LIN {X 0,Y 389.077,Z 656.988,A -85,B 0,C 180,E1 10601.483,E2 10601.483} C_VEL
LIN {X 0,Y 373.239,Z 818.988,A -85,B 0,C 180,E1 10598.992,E2 10598.992} C_VEL
LIN {X 0,Y 369.039,Z 845.316,A -85,B 0,C 180,E1 10598.451,E2 10598.451} C_VEL
LIN {X 0,Y 364.552,Z 865.956,A -85,B 0,C 180,E1 10597.891,E2 10597.891} C_VEL
LIN {X 0,Y 357.971,Z 890.119,A -85,B 0,C 180,E1 10597.055,E2 10597.055} C_VEL
LIN {X 0,Y 350.974,Z 911.054,A -85,B 0,C 180,E1 10596.135,E2 10596.135} C_VEL
LIN {X 0,Y 342.625,Z 932.727,A -85,B 0,C 180,E1 10594.966,E2 10594.966} C_VEL
LIN {X 0,Y 332.858,Z 954.168,A -85,B 0,C 180,E1 10593.532,E2 10593.532} C_VEL
LIN {X 0,Y 322.694,Z 974.134,A -85,B 0,C 180,E1 10591.902,E2 10591.902} C_VEL
LIN {X 0,Y 311.477,Z 993.542,A -85,B 0,C 180,E1 10589.948,E2 10589.948} C_VEL
LIN {X 0,Y 300.928,Z 1010.196,A -85,B 0,C 180,E1 10587.918,E2 10587.918} C_VEL
LIN {X 0,Y 287.781,Z 1029.047,A -85,B 0,C 180,E1 10585.083,E2 10585.083} C_VEL
LIN {X 0,Y 276.633,Z 1043.791,A -85,B 0,C 180,E1 10582.333,E2 10582.333} C_VEL
LIN {X 0,Y 263.742,Z 1059.682,A -85,B 0,C 180,E1 10578.647,E2 10578.647} C_VEL
LIN {X 0,Y 253.035,Z 1072.129,A -85,B 0,C 180,E1 10575.019,E2 10575.019} C_VEL
LIN {X 0,Y 241.418,Z 1085.134,A -85,B 0,C 180,E1 10570.249,E2 10570.249} C_VEL
LIN {X 0,Y 232.232,Z 1095.159,A -85,B 0,C 180,E1 10565.539,E2 10565.539} C_VEL
LIN {X 0,Y 223.527,Z 1104.789,A -85,B 0,C 180,E1 10559.771,E2 10559.771} C_VEL
LIN {X 0,Y 217.336,Z 1111.9,A -85,B 0,C 180,E1 10554.171,E2 10554.171} C_VEL
LIN {X 0,Y 212.563,Z 1118.125,A -85,B 0,C 180,E1 10547.804,E2 10547.804} C_VEL
LIN {X 0,Y 209.773,Z 1122.382,A -85,B 0,C 180,E1 10541.548,E2 10541.548} C_VEL
LIN {X 0,Y 208.571,Z 1124.988,A -85,B 0,C 180,E1 10536.054,E2 10536.054} C_VEL
LIN {X 0,Y 208.165,Z 1126.701,A -85,B 0,C 180,E1 10530,E2 10530} C_VEL
LIN {X 0,Y 208.154,Z 1127.046,A -85,B 0,C 180,E1 10524.21,E2 10524.21} C_VEL
LIN {X 0,Y 208.486,Z 1126.397,A -85,B 0,C 180,E1 10518.94,E2 10518.94} C_VEL
LIN {X 0,Y 209.585,Z 1124.699,A -85,B 0,C 180,E1 10513.366,E2 10513.366} C_VEL
LIN {X 0,Y 212.305,Z 1121.48,A -85,B 0,C 180,E1 10506.989,E2 10506.989} C_VEL
LIN {X 0,Y 217.097,Z 1116.332,A -85,B 0,C 180,E1 10500.474,E2 10500.474} C_VEL
LIN {X 0,Y 223.889,Z 1109.804,A -85,B 0,C 180,E1 10494.372,E2 10494.372} C_VEL
LIN {X 0,Y 232.384,Z 1101.701,A -85,B 0,C 180,E1 10488.828,E2 10488.828} C_VEL
LIN {X 0,Y 241.918,Z 1092.689,A -85,B 0,C 180,E1 10484.013,E2 10484.013} C_VEL
LIN {X 0,Y 254.032,Z 1080.851,A -85,B 0,C 180,E1 10479.158,E2 10479.158} C_VEL
LIN {X 0,Y 265.219,Z 1069.449,A -85,B 0,C 180,E1 10475.478,E2 10475.478} C_VEL
LIN {X 0,Y 278.682,Z 1054.854,A -85,B 0,C 180,E1 10471.751,E2 10471.751} C_VEL
LIN {X 0,Y 290.339,Z 1041.264,A -85,B 0,C 180,E1 10468.985,E2 10468.985} C_VEL
LIN {X 0,Y 303.745,Z 1024.447,A -85,B 0,C 180,E1 10466.207,E2 10466.207} C_VEL
LIN {X 0,Y 315.589,Z 1008.029,A -85,B 0,C 180,E1 10464.034,E2 10464.034} C_VEL
LIN {X 0,Y 327.873,Z 989.488,A -85,B 0,C 180,E1 10462.014,E2 10462.014} C_VEL
LIN {X 0,Y 339.512,Z 969.544,A -85,B 0,C 180,E1 10460.266,E2 10460.266} C_VEL
LIN {X 0,Y 349.337,Z 950.846,A -85,B 0,C 180,E1 10458.919,E2 10458.919} C_VEL
LIN {X 0,Y 359.347,Z 928.996,A -85,B 0,C 180,E1 10457.633,E2 10457.633} C_VEL
LIN {X 0,Y 366.943,Z 909.841,A -85,B 0,C 180,E1 10456.702,E2 10456.702} C_VEL
LIN {X 0,Y 374.785,Z 886.816,A -85,B 0,C 180,E1 10455.791,E2 10455.791} C_VEL
LIN {X 0,Y 381.061,Z 863.843,A -85,B 0,C 180,E1 10455.085,E2 10455.085} C_VEL
LIN {X 0,Y 386.288,Z 839.912,A -85,B 0,C 180,E1 10454.513,E2 10454.513} C_VEL
LIN {X 0,Y 389.922,Z 815.583,A -85,B 0,C 180,E1 10454.078,E2 10454.078} C_VEL
LIN {X 0,Y 404.87,Z 668.819,A -85,B 0,C 180,E1 10451.908,E2 10451.908} C_VEL
LIN {X 0,Y 401.866,Z 662.718,A -85,B 0,C 180,E1 10449.38,E2 10449.38} C_VEL
LIN {X 0,Y 400.205,Z 659.502,A -85,B 0,C 180,E1 10447.682,E2 10447.682} C_VEL
LIN {X 0,Y 398.698,Z 656.415,A -85,B 0,C 180,E1 10445.757,E2 10445.757} C_VEL
LIN {X 0,Y 396.955,Z 652.484,A -85,B 0,C 180,E1 10442.31,E2 10442.31} C_VEL
LIN {X 0,Y 396.309,Z 651.938,A -85,B 0,C 180,E1 10437.686,E2 10437.686} C_VEL
LIN {X 0,Y 397.092,Z 652.674,A -85,B 0,C 180,E1 10434.799,E2 10434.799} C_VEL
LIN {X 0,Y 397.231,Z 653.236,A -85,B 0,C 180,E1 10434.385,E2 10434.385} C_VEL
LIN {X 0,Y 397.569,Z 655.643,A -85,B 0,C 180,E1 10433.318,E2 10433.318} C_VEL
LIN {X 0,Y 398.682,Z 666,A -85,B 0,C 180,E1 10430.456,E2 10430.456} C_VEL
LIN {X 0,Y 399.282,Z 667.678,A -85,B 0,C 180,E1 10429.696,E2 10429.696} C_VEL
LIN {X 0,Y 401.751,Z 672.925,A -85,B 0,C 180,E1 10427.239,E2 10427.239} C_VEL
LIN {X 0,Y 402.563,Z 675.356,A -85,B 0,C 180,E1 10426.485,E2 10426.485} C_VEL
LIN {X 0,Y 386.785,Z 826.745,A -85,B 0,C 180,E1 10424.281,E2 10424.281} C_VEL
LIN {X 0,Y 382.278,Z 853.306,A -85,B 0,C 180,E1 10423.81,E2 10423.81} C_VEL
LIN {X 0,Y 377.108,Z 875.277,A -85,B 0,C 180,E1 10423.339,E2 10423.339} C_VEL
LIN {X 0,Y 369.772,Z 899.868,A -85,B 0,C 180,E1 10422.658,E2 10422.658} C_VEL
LIN {X 0,Y 362.204,Z 920.785,A -85,B 0,C 180,E1 10421.909,E2 10421.909} C_VEL
LIN {X 0,Y 352.874,Z 943.017,A -85,B 0,C 180,E1 10420.908,E2 10420.908} C_VEL
LIN {X 0,Y 343.111,Z 962.976,A -85,B 0,C 180,E1 10419.78,E2 10419.78} C_VEL
LIN {X 0,Y 332.272,Z 982.798,A -85,B 0,C 180,E1 10418.414,E2 10418.414} C_VEL
LIN {X 0,Y 320.029,Z 1002.552,A -85,B 0,C 180,E1 10416.718,E2 10416.718} C_VEL
LIN {X 0,Y 308.525,Z 1019.414,A -85,B 0,C 180,E1 10414.935,E2 10414.935} C_VEL
LIN {X 0,Y 294.339,Z 1038.307,A -85,B 0,C 180,E1 10412.454,E2 10412.454} C_VEL
LIN {X 0,Y 281.858,Z 1053.497,A -85,B 0,C 180,E1 10409.95,E2 10409.95} C_VEL
LIN {X 0,Y 267.962,Z 1069.274,A -85,B 0,C 180,E1 10406.705,E2 10406.705} C_VEL
LIN {X 0,Y 255.148,Z 1082.75,A -85,B 0,C 180,E1 10403.16,E2 10403.16} C_VEL
LIN {X 0,Y 242.608,Z 1095.445,A -85,B 0,C 180,E1 10398.958,E2 10398.958} C_VEL
LIN {X 0,Y 231.059,Z 1106.532,A -85,B 0,C 180,E1 10394.164,E2 10394.164} C_VEL
LIN {X 0,Y 220.814,Z 1116.462,A -85,B 0,C 180,E1 10388.674,E2 10388.674} C_VEL
LIN {X 0,Y 212.27,Z 1124.783,A -85,B 0,C 180,E1 10382.479,E2 10382.479} C_VEL
LIN {X 0,Y 206.062,Z 1131.495,A -85,B 0,C 180,E1 10375.895,E2 10375.895} C_VEL
LIN {X 0,Y 202.161,Z 1136.355,A -85,B 0,C 180,E1 10369.053,E2 10369.053} C_VEL
LIN {X 0,Y 200.522,Z 1139.217,A -85,B 0,C 180,E1 10363.26,E2 10363.26} C_VEL
LIN {X 0,Y 200.045,Z 1141.13,A -85,B 0,C 180,E1 10356.89,E2 10356.89} C_VEL
LIN {X 0,Y 200.113,Z 1141.605,A -85,B 0,C 180,E1 10351.432,E2 10351.432} C_VEL
LIN {X 0,Y 200.082,Z 1141.072,A -85,B 0,C 180,E1 10346.275,E2 10346.275} C_VEL
LIN {X 0,Y 200.105,Z 1139.478,A -85,B 0,C 180,E1 10340.799,E2 10340.799} C_VEL
LIN {X 0,Y 200.858,Z 1136.684,A -85,B 0,C 180,E1 10334.997,E2 10334.997} C_VEL
LIN {X 0,Y 203.257,Z 1132.107,A -85,B 0,C 180,E1 10328.349,E2 10328.349} C_VEL
LIN {X 0,Y 207.889,Z 1125.467,A -85,B 0,C 180,E1 10321.565,E2 10321.565} C_VEL
LIN {X 0,Y 214.178,Z 1117.89,A -85,B 0,C 180,E1 10315.605,E2 10315.605} C_VEL
LIN {X 0,Y 222.875,Z 1108.056,A -85,B 0,C 180,E1 10309.701,E2 10309.701} C_VEL
LIN {X 0,Y 231.964,Z 1098.075,A -85,B 0,C 180,E1 10304.986,E2 10304.986} C_VEL
LIN {X 0,Y 244.099,Z 1084.603,A -85,B 0,C 180,E1 10300.004,E2 10300.004} C_VEL
LIN {X 0,Y 254.771,Z 1072.356,A -85,B 0,C 180,E1 10296.432,E2 10296.432} C_VEL
LIN {X 0,Y 267.773,Z 1056.749,A -85,B 0,C 180,E1 10292.782,E2 10292.782} C_VEL
LIN {X 0,Y 279.395,Z 1041.739,A -85,B 0,C 180,E1 10289.995,E2 10289.995} C_VEL
LIN {X 0,Y 292.125,Z 1024.23,A -85,B 0,C 180,E1 10287.349,E2 10287.349} C_VEL
LIN {X 0,Y 304.257,Z 1005.693,A -85,B 0,C 180,E1 10285.124,E2 10285.124} C_VEL
LIN {X 0,Y 315.234,Z 987.407,A -85,B 0,C 180,E1 10283.325,E2 10283.325} C_VEL
LIN {X 0,Y 326.531,Z 966.324,A -85,B 0,C 180,E1 10281.663,E2 10281.663} C_VEL
LIN {X 0,Y 336.004,Z 946.38,A -85,B 0,C 180,E1 10280.382,E2 10280.382} C_VEL
LIN {X 0,Y 345.665,Z 922.993,A -85,B 0,C 180,E1 10279.186,E2 10279.186} C_VEL
LIN {X 0,Y 352.927,Z 902.419,A -85,B 0,C 180,E1 10278.358,E2 10278.358} C_VEL
LIN {X 0,Y 360.033,Z 878.466,A -85,B 0,C 180,E1 10277.598,E2 10277.598} C_VEL
LIN {X 0,Y 365.3,Z 855.714,A -85,B 0,C 180,E1 10277.045,E2 10277.045} C_VEL
LIN {X 0,Y 369.595,Z 830.946,A -85,B 0,C 180,E1 10276.554,E2 10276.554} C_VEL
LIN {X 0,Y 375.172,Z 776.826,A -85,B 0,C 180,E1 10275.706,E2 10275.706} C_VEL
LIN {X 0,Y 386.379,Z 662.671,A -85,B 0,C 180,E1 10273.975,E2 10273.975} C_VEL
LIN {X 0,Y 384.218,Z 657.456,A -85,B 0,C 180,E1 10272.398,E2 10272.398} C_VEL
LIN {X 0,Y 380.921,Z 650.9,A -85,B 0,C 180,E1 10269.671,E2 10269.671} C_VEL
LIN {X 0,Y 378.814,Z 646.848,A -85,B 0,C 180,E1 10267.508,E2 10267.508} C_VEL
LIN {X 0,Y 377.258,Z 643.74,A -85,B 0,C 180,E1 10265.475,E2 10265.475} C_VEL
LIN {X 0,Y 375.486,Z 639.736,A -85,B 0,C 180,E1 10261.831,E2 10261.831} C_VEL
LIN {X 0,Y 374.913,Z 639.355,A -85,B 0,C 180,E1 10256.789,E2 10256.789} C_VEL
LIN {X 0,Y 375.595,Z 640.112,A -85,B 0,C 180,E1 10254.271,E2 10254.271} C_VEL
LIN {X 0,Y 377.781,Z 644.756,A -85,B 0,C 180,E1 10250.247,E2 10250.247} C_VEL
LIN {X 0,Y 380.132,Z 649.399,A -85,B 0,C 180,E1 10247.544,E2 10247.544} C_VEL
LIN {X 0,Y 382.994,Z 654.95,A -85,B 0,C 180,E1 10245.01,E2 10245.01} C_VEL
LIN {X 0,Y 386.347,Z 662.03,A -85,B 0,C 180,E1 10242.546,E2 10242.546} C_VEL
LIN {X 0,Y 370.657,Z 819.269,A -85,B 0,C 180,E1 10240.158,E2 10240.158} C_VEL
LIN {X 0,Y 366.382,Z 845.61,A -85,B 0,C 180,E1 10239.627,E2 10239.627} C_VEL
LIN {X 0,Y 361.82,Z 866.249,A -85,B 0,C 180,E1 10239.078,E2 10239.078} C_VEL
LIN {X 0,Y 355.206,Z 890.16,A -85,B 0,C 180,E1 10238.27,E2 10238.27} C_VEL
LIN {X 0,Y 347.96,Z 911.47,A -85,B 0,C 180,E1 10237.352,E2 10237.352} C_VEL
LIN {X 0,Y 339.387,Z 933.291,A -85,B 0,C 180,E1 10236.195,E2 10236.195} C_VEL
LIN {X 0,Y 329.373,Z 954.809,A -85,B 0,C 180,E1 10234.777,E2 10234.777} C_VEL
LIN {X 0,Y 318.967,Z 974.805,A -85,B 0,C 180,E1 10233.166,E2 10233.166} C_VEL
LIN {X 0,Y 307.443,Z 994.243,A -85,B 0,C 180,E1 10231.227,E2 10231.227} C_VEL
LIN {X 0,Y 296.734,Z 1010.729,A -85,B 0,C 180,E1 10229.234,E2 10229.234} C_VEL
LIN {X 0,Y 283.243,Z 1029.541,A -85,B 0,C 180,E1 10226.421,E2 10226.421} C_VEL
LIN {X 0,Y 271.77,Z 1044.267,A -85,B 0,C 180,E1 10223.682,E2 10223.682} C_VEL
LIN {X 0,Y 258.461,Z 1060.127,A -85,B 0,C 180,E1 10219.995,E2 10219.995} C_VEL
LIN {X 0,Y 247.367,Z 1072.561,A -85,B 0,C 180,E1 10216.348,E2 10216.348} C_VEL
LIN {X 0,Y 235.281,Z 1085.54,A -85,B 0,C 180,E1 10211.527,E2 10211.527} C_VEL
LIN {X 0,Y 226.096,Z 1095.105,A -85,B 0,C 180,E1 10206.974,E2 10206.974} C_VEL
LIN {X 0,Y 217.212,Z 1104.472,A -85,B 0,C 180,E1 10201.344,E2 10201.344} C_VEL
LIN {X 0,Y 210.232,Z 1111.963,A -85,B 0,C 180,E1 10195.344,E2 10195.344} C_VEL
LIN {X 0,Y 205.225,Z 1118.003,A -85,B 0,C 180,E1 10189.053,E2 10189.053} C_VEL
LIN {X 0,Y 201.995,Z 1122.551,A -85,B 0,C 180,E1 10182.29,E2 10182.29} C_VEL
LIN {X 0,Y 200.645,Z 1125.189,A -85,B 0,C 180,E1 10176.582,E2 10176.582} C_VEL
LIN {X 0,Y 200.184,Z 1126.867,A -85,B 0,C 180,E1 10170.572,E2 10170.572} C_VEL
LIN {X 0,Y 200.146,Z 1127.368,A -85,B 0,C 180,E1 10164.553,E2 10164.553} C_VEL
LIN {X 0,Y 200.509,Z 1126.734,A -85,B 0,C 180,E1 10158.785,E2 10158.785} C_VEL
LIN {X 0,Y 201.683,Z 1125.072,A -85,B 0,C 180,E1 10152.992,E2 10152.992} C_VEL
LIN {X 0,Y 204.58,Z 1121.892,A -85,B 0,C 180,E1 10146.373,E2 10146.373} C_VEL
LIN {X 0,Y 209.663,Z 1116.815,A -85,B 0,C 180,E1 10139.634,E2 10139.634} C_VEL
LIN {X 0,Y 216.332,Z 1110.749,A -85,B 0,C 180,E1 10133.728,E2 10133.728} C_VEL
LIN {X 0,Y 225.749,Z 1102.302,A -85,B 0,C 180,E1 10127.682,E2 10127.682} C_VEL
LIN {X 0,Y 235.188,Z 1093.784,A -85,B 0,C 180,E1 10123.008,E2 10123.008} C_VEL
LIN {X 0,Y 248.282,Z 1081.583,A -85,B 0,C 180,E1 10117.876,E2 10117.876} C_VEL
LIN {X 0,Y 259.85,Z 1070.229,A -85,B 0,C 180,E1 10114.176,E2 10114.176} C_VEL
LIN {X 0,Y 273.728,Z 1055.738,A -85,B 0,C 180,E1 10110.449,E2 10110.449} C_VEL
LIN {X 0,Y 285.701,Z 1042.207,A -85,B 0,C 180,E1 10107.693,E2 10107.693} C_VEL
LIN {X 0,Y 299.404,Z 1025.573,A -85,B 0,C 180,E1 10104.946,E2 10104.946} C_VEL
LIN {X 0,Y 312.128,Z 1008.359,A -85,B 0,C 180,E1 10102.691,E2 10102.691} C_VEL
LIN {X 0,Y 324.234,Z 990.491,A -85,B 0,C 180,E1 10100.772,E2 10100.772} C_VEL
LIN {X 0,Y 336.332,Z 970.282,A -85,B 0,C 180,E1 10099.021,E2 10099.021} C_VEL
LIN {X 0,Y 346.358,Z 951.586,A -85,B 0,C 180,E1 10097.698,E2 10097.698} C_VEL
LIN {X 0,Y 357.078,Z 928.575,A -85,B 0,C 180,E1 10096.375,E2 10096.375} C_VEL
LIN {X 0,Y 364.695,Z 909.63,A -85,B 0,C 180,E1 10095.481,E2 10095.481} C_VEL
LIN {X 0,Y 372.939,Z 885.495,A -85,B 0,C 180,E1 10094.56,E2 10094.56} C_VEL
LIN {X 0,Y 379.007,Z 863.476,A -85,B 0,C 180,E1 10093.906,E2 10093.906} C_VEL
LIN {X 0,Y 384.313,Z 839.198,A -85,B 0,C 180,E1 10093.347,E2 10093.347} C_VEL
LIN {X 0,Y 387.882,Z 815.546,A -85,B 0,C 180,E1 10092.935,E2 10092.935} C_VEL
LIN {X 0,Y 402.529,Z 674.462,A -85,B 0,C 180,E1 10090.882,E2 10090.882} C_VEL
LIN {X 0,Y 399.548,Z 668.179,A -85,B 0,C 180,E1 10088.056,E2 10088.056} C_VEL
LIN {X 0,Y 397.512,Z 664.147,A -85,B 0,C 180,E1 10085.485,E2 10085.485} C_VEL
LIN {X 0,Y 395.923,Z 660.389,A -85,B 0,C 180,E1 10082.171,E2 10082.171} C_VEL
LIN {X 0,Y 395.335,Z 659.88,A -85,B 0,C 180,E1 10077.681,E2 10077.681} C_VEL
LIN {X 0,Y 396.102,Z 660.773,A -85,B 0,C 180,E1 10074.786,E2 10074.786} C_VEL
LIN {X 0,Y 398.074,Z 665.191,A -85,B 0,C 180,E1 10071.186,E2 10071.186} C_VEL
LIN {X 0,Y 399.282,Z 667.678,A -85,B 0,C 180,E1 10069.696,E2 10069.696} C_VEL
LIN {X 0,Y 399.859,Z 669.792,A -85,B 0,C 180,E1 10068.972,E2 10068.972} C_VEL
LIN {X 0,Y 400.217,Z 673.868,A -85,B 0,C 180,E1 10068.278,E2 10068.278} C_VEL
LIN {X 0,Y 400.253,Z 679.11,A -85,B 0,C 180,E1 10067.758,E2 10067.758} C_VEL
LIN {X 0,Y 399.966,Z 684.336,A -85,B 0,C 180,E1 10067.491,E2 10067.491} C_VEL
LIN {X 0,Y 399.817,Z 685.9,A -85,B 0,C 180,E1 10067.457,E2 10067.457} C_VEL
LIN {X 0,Y 384.869,Z 826.589,A -85,B 0,C 180,E1 10065.439,E2 10065.439} C_VEL
LIN {X 0,Y 380.298,Z 853.099,A -85,B 0,C 180,E1 10064.98,E2 10064.98} C_VEL
LIN {X 0,Y 375.076,Z 875.003,A -85,B 0,C 180,E1 10064.525,E2 10064.525} C_VEL
LIN {X 0,Y 367.463,Z 900.11,A -85,B 0,C 180,E1 10063.851,E2 10063.851} C_VEL
LIN {X 0,Y 359.939,Z 920.591,A -85,B 0,C 180,E1 10063.138,E2 10063.138} C_VEL
LIN {X 0,Y 350.323,Z 943.101,A -85,B 0,C 180,E1 10062.153,E2 10062.153} C_VEL
LIN {X 0,Y 340.403,Z 963.023,A -85,B 0,C 180,E1 10061.056,E2 10061.056} C_VEL
LIN {X 0,Y 328.958,Z 983.547,A -85,B 0,C 180,E1 10059.671,E2 10059.671} C_VEL
LIN {X 0,Y 316.678,Z 1002.842,A -85,B 0,C 180,E1 10058.038,E2 10058.038} C_VEL
LIN {X 0,Y 304.36,Z 1020.464,A -85,B 0,C 180,E1 10056.197,E2 10056.197} C_VEL
LIN {X 0,Y 289.871,Z 1039.135,A -85,B 0,C 180,E1 10053.748,E2 10053.748} C_VEL
LIN {X 0,Y 277.099,Z 1054.228,A -85,B 0,C 180,E1 10051.265,E2 10051.265} C_VEL
LIN {X 0,Y 262.14,Z 1070.537,A -85,B 0,C 180,E1 10047.864,E2 10047.864} C_VEL
LIN {X 0,Y 249.695,Z 1083.167,A -85,B 0,C 180,E1 10044.504,E2 10044.504} C_VEL
LIN {X 0,Y 236.086,Z 1096.303,A -85,B 0,C 180,E1 10040.049,E2 10040.049} C_VEL
LIN {X 0,Y 224.674,Z 1106.797,A -85,B 0,C 180,E1 10035.403,E2 10035.403} C_VEL
LIN {X 0,Y 213.98,Z 1116.629,A -85,B 0,C 180,E1 10029.805,E2 10029.805} C_VEL
LIN {X 0,Y 205.335,Z 1124.55,A -85,B 0,C 180,E1 10023.72,E2 10023.72} C_VEL
LIN {X 0,Y 198.673,Z 1131.253,A -85,B 0,C 180,E1 10016.934,E2 10016.934} C_VEL
LIN {X 0,Y 194.385,Z 1136.161,A -85,B 0,C 180,E1 10009.723,E2 10009.723} C_VEL
LIN {X 0,Y 192.556,Z 1139.07,A -85,B 0,C 180,E1 10003.513,E2 10003.513} C_VEL
LIN {X 0,Y 192.048,Z 1140.945,A -85,B 0,C 180,E1 9996.577,E2 9996.577} C_VEL
LIN {X 0,Y 192.121,Z 1141.274,A -85,B 0,C 180,E1 9990.895,E2 9990.895} C_VEL
LIN {X 0,Y 192.078,Z 1140.703,A -85,B 0,C 180,E1 9985.821,E2 9985.821} C_VEL
LIN {X 0,Y 192.142,Z 1139.049,A -85,B 0,C 180,E1 9980.112,E2 9980.112} C_VEL
LIN {X 0,Y 192.988,Z 1136.362,A -85,B 0,C 180,E1 9974.37,E2 9974.37} C_VEL
LIN {X 0,Y 195.632,Z 1131.773,A -85,B 0,C 180,E1 9967.46,E2 9967.46} C_VEL
LIN {X 0,Y 200.653,Z 1125.111,A -85,B 0,C 180,E1 9960.44,E2 9960.44} C_VEL
LIN {X 0,Y 207.38,Z 1117.523,A -85,B 0,C 180,E1 9954.309,E2 9954.309} C_VEL
LIN {X 0,Y 216.52,Z 1107.744,A -85,B 0,C 180,E1 9948.318,E2 9948.318} C_VEL
LIN {X 0,Y 226.114,Z 1097.716,A -85,B 0,C 180,E1 9943.513,E2 9943.513} C_VEL
LIN {X 0,Y 238.835,Z 1084.176,A -85,B 0,C 180,E1 9938.474,E2 9938.474} C_VEL
LIN {X 0,Y 250.571,Z 1071.2,A -85,B 0,C 180,E1 9934.711,E2 9934.711} C_VEL
LIN {X 0,Y 264.956,Z 1054.323,A -85,B 0,C 180,E1 9930.88,E2 9930.88} C_VEL
LIN {X 0,Y 276.82,Z 1039.367,A -85,B 0,C 180,E1 9928.195,E2 9928.195} C_VEL
LIN {X 0,Y 290.783,Z 1020.259,A -85,B 0,C 180,E1 9925.457,E2 9925.457} C_VEL
LIN {X 0,Y 302.045,Z 1003.294,A -85,B 0,C 180,E1 9923.51,E2 9923.51} C_VEL
LIN {X 0,Y 314.123,Z 983.325,A -85,B 0,C 180,E1 9921.647,E2 9921.647} C_VEL
LIN {X 0,Y 324.853,Z 963.234,A -85,B 0,C 180,E1 9920.151,E2 9920.151} C_VEL
LIN {X 0,Y 334.956,Z 942.068,A -85,B 0,C 180,E1 9918.863,E2 9918.863} C_VEL
LIN {X 0,Y 343.939,Z 919.952,A -85,B 0,C 180,E1 9917.805,E2 9917.805} C_VEL
LIN {X 0,Y 351.763,Z 897.705,A -85,B 0,C 180,E1 9916.959,E2 9916.959} C_VEL
LIN {X 0,Y 358.664,Z 873.459,A -85,B 0,C 180,E1 9916.257,E2 9916.257} C_VEL
LIN {X 0,Y 363.79,Z 850.822,A -85,B 0,C 180,E1 9915.744,E2 9915.744} C_VEL
LIN {X 0,Y 367.843,Z 825.226,A -85,B 0,C 180,E1 9915.274,E2 9915.274} C_VEL
LIN {X 0,Y 383.786,Z 667.615,A -85,B 0,C 180,E1 9912.896,E2 9912.896} C_VEL
LIN {X 0,Y 382.053,Z 663.645,A -85,B 0,C 180,E1 9911.549,E2 9911.549} C_VEL
LIN {X 0,Y 379.288,Z 658.009,A -85,B 0,C 180,E1 9909.101,E2 9909.101} C_VEL
LIN {X 0,Y 377.498,Z 654.416,A -85,B 0,C 180,E1 9907.151,E2 9907.151} C_VEL
LIN {X 0,Y 376.065,Z 651.473,A -85,B 0,C 180,E1 9905.187,E2 9905.187} C_VEL
LIN {X 0,Y 374.453,Z 647.647,A -85,B 0,C 180,E1 9901.683,E2 9901.683} C_VEL
LIN {X 0,Y 373.963,Z 647.319,A -85,B 0,C 180,E1 9896.628,E2 9896.628} C_VEL
LIN {X 0,Y 374.54,Z 647.918,A -85,B 0,C 180,E1 9894.485,E2 9894.485} C_VEL
LIN {X 0,Y 376.627,Z 652.584,A -85,B 0,C 180,E1 9890.449,E2 9890.449} C_VEL
LIN {X 0,Y 378.842,Z 657.104,A -85,B 0,C 180,E1 9887.81,E2 9887.81} C_VEL
LIN {X 0,Y 381.562,Z 662.602,A -85,B 0,C 180,E1 9885.313,E2 9885.313} C_VEL
LIN {X 0,Y 383.713,Z 667.446,A -85,B 0,C 180,E1 9883.618,E2 9883.618} C_VEL
LIN {X 0,Y 368.221,Z 819.606,A -85,B 0,C 180,E1 9881.339,E2 9881.339} C_VEL
LIN {X 0,Y 363.882,Z 845.895,A -85,B 0,C 180,E1 9880.82,E2 9880.82} C_VEL
LIN {X 0,Y 359.234,Z 866.58,A -85,B 0,C 180,E1 9880.282,E2 9880.282} C_VEL
LIN {X 0,Y 352.338,Z 891.006,A -85,B 0,C 180,E1 9879.472,E2 9879.472} C_VEL
LIN {X 0,Y 345.074,Z 911.975,A -85,B 0,C 180,E1 9878.586,E2 9878.586} C_VEL
LIN {X 0,Y 336.31,Z 933.844,A -85,B 0,C 180,E1 9877.447,E2 9877.447} C_VEL
LIN {X 0,Y 326.449,Z 954.651,A -85,B 0,C 180,E1 9876.105,E2 9876.105} C_VEL
LIN {X 0,Y 316.492,Z 973.458,A -85,B 0,C 180,E1 9874.63,E2 9874.63} C_VEL
LIN {X 0,Y 304.419,Z 993.614,A -85,B 0,C 180,E1 9872.684,E2 9872.684} C_VEL
LIN {X 0,Y 293.442,Z 1010.17,A -85,B 0,C 180,E1 9870.729,E2 9870.729} C_VEL
LIN {X 0,Y 279.579,Z 1029.125,A -85,B 0,C 180,E1 9867.953,E2 9867.953} C_VEL
LIN {X 0,Y 267.742,Z 1043.915,A -85,B 0,C 180,E1 9865.245,E2 9865.245} C_VEL
LIN {X 0,Y 253.964,Z 1059.886,A -85,B 0,C 180,E1 9861.582,E2 9861.582} C_VEL
LIN {X 0,Y 242.418,Z 1072.371,A -85,B 0,C 180,E1 9857.94,E2 9857.94} C_VEL
LIN {X 0,Y 230.302,Z 1084.94,A -85,B 0,C 180,E1 9853.313,E2 9853.313} C_VEL
LIN {X 0,Y 220.112,Z 1095.051,A -85,B 0,C 180,E1 9848.488,E2 9848.488} C_VEL
LIN {X 0,Y 210.696,Z 1104.492,A -85,B 0,C 180,E1 9842.752,E2 9842.752} C_VEL
LIN {X 0,Y 202.943,Z 1112.319,A -85,B 0,C 180,E1 9836.323,E2 9836.323} C_VEL
LIN {X 0,Y 197.517,Z 1118.465,A -85,B 0,C 180,E1 9829.679,E2 9829.679} C_VEL
LIN {X 0,Y 194.144,Z 1122.873,A -85,B 0,C 180,E1 9822.795,E2 9822.795} C_VEL
LIN {X 0,Y 192.686,Z 1125.499,A -85,B 0,C 180,E1 9816.855,E2 9816.855} C_VEL
LIN {X 0,Y 192.19,Z 1127.167,A -85,B 0,C 180,E1 9810.596,E2 9810.596} C_VEL
LIN {X 0,Y 192.149,Z 1127.669,A -85,B 0,C 180,E1 9804.625,E2 9804.625} C_VEL
LIN {X 0,Y 192.532,Z 1127.07,A -85,B 0,C 180,E1 9798.618,E2 9798.618} C_VEL
LIN {X 0,Y 193.789,Z 1125.444,A -85,B 0,C 180,E1 9792.587,E2 9792.587} C_VEL
LIN {X 0,Y 196.704,Z 1122.455,A -85,B 0,C 180,E1 9786.005,E2 9786.005} C_VEL
LIN {X 0,Y 202.278,Z 1117.298,A -85,B 0,C 180,E1 9778.733,E2 9778.733} C_VEL
LIN {X 0,Y 208.959,Z 1111.566,A -85,B 0,C 180,E1 9772.92,E2 9772.92} C_VEL
LIN {X 0,Y 219.211,Z 1102.903,A -85,B 0,C 180,E1 9766.468,E2 9766.468} C_VEL
LIN {X 0,Y 229.062,Z 1094.427,A -85,B 0,C 180,E1 9761.717,E2 9761.717} C_VEL
LIN {X 0,Y 242.062,Z 1082.882,A -85,B 0,C 180,E1 9756.74,E2 9756.74} C_VEL
LIN {X 0,Y 253.968,Z 1071.638,A -85,B 0,C 180,E1 9753.007,E2 9753.007} C_VEL
LIN {X 0,Y 267.52,Z 1058.146,A -85,B 0,C 180,E1 9749.44,E2 9749.44} C_VEL
LIN {X 0,Y 281.214,Z 1043.152,A -85,B 0,C 180,E1 9746.36,E2 9746.36} C_VEL
LIN {X 0,Y 294.859,Z 1027.081,A -85,B 0,C 180,E1 9743.709,E2 9743.709} C_VEL
LIN {X 0,Y 308.25,Z 1009.51,A -85,B 0,C 180,E1 9741.414,E2 9741.414} C_VEL
LIN {X 0,Y 320.025,Z 992.566,A -85,B 0,C 180,E1 9739.607,E2 9739.607} C_VEL
LIN {X 0,Y 332.916,Z 971.716,A -85,B 0,C 180,E1 9737.807,E2 9737.807} C_VEL
LIN {X 0,Y 342.875,Z 953.59,A -85,B 0,C 180,E1 9736.538,E2 9736.538} C_VEL
LIN {X 0,Y 353.825,Z 930.858,A -85,B 0,C 180,E1 9735.237,E2 9735.237} C_VEL
LIN {X 0,Y 361.892,Z 911.284,A -85,B 0,C 180,E1 9734.323,E2 9734.323} C_VEL
LIN {X 0,Y 370.104,Z 888.109,A -85,B 0,C 180,E1 9733.444,E2 9733.444} C_VEL
LIN {X 0,Y 376.708,Z 864.713,A -85,B 0,C 180,E1 9732.757,E2 9732.757} C_VEL
LIN {X 0,Y 382.095,Z 840.871,A -85,B 0,C 180,E1 9732.214,E2 9732.214} C_VEL
LIN {X 0,Y 385.882,Z 816.421,A -85,B 0,C 180,E1 9731.794,E2 9731.794} C_VEL
LIN {X 0,Y 400.271,Z 680.226,A -85,B 0,C 180,E1 9729.82,E2 9729.82} C_VEL
LIN {X 0,Y 397.908,Z 675.214,A -85,B 0,C 180,E1 9727.363,E2 9727.363} C_VEL
LIN {X 0,Y 396.336,Z 671.876,A -85,B 0,C 180,E1 9725.211,E2 9725.211} C_VEL
LIN {X 0,Y 394.894,Z 668.294,A -85,B 0,C 180,E1 9722.032,E2 9722.032} C_VEL
LIN {X 0,Y 394.377,Z 667.84,A -85,B 0,C 180,E1 9717.53,E2 9717.53} C_VEL
LIN {X 0,Y 395.067,Z 668.674,A -85,B 0,C 180,E1 9714.918,E2 9714.918} C_VEL
LIN {X 0,Y 396.978,Z 673.142,A -85,B 0,C 180,E1 9711.308,E2 9711.308} C_VEL
LIN {X 0,Y 398.945,Z 677.376,A -85,B 0,C 180,E1 9708.946,E2 9708.946} C_VEL
LIN {X 0,Y 400.374,Z 680.559,A -85,B 0,C 180,E1 9707.538,E2 9707.538} C_VEL
LIN {X 0,Y 399.817,Z 685.9,A -85,B 0,C 180,E1 9707.457,E2 9707.457} C_VEL
LIN {X 0,Y 398.811,Z 693.597,A -85,B 0,C 180,E1 9707.488,E2 9707.488} C_VEL
LIN {X 0,Y 395.427,Z 714.159,A -85,B 0,C 180,E1 9708.09,E2 9708.09} C_VEL
LIN {X 0,Y 394.58,Z 720.765,A -85,B 0,C 180,E1 9708.107,E2 9708.107} C_VEL
LIN {X 0,Y 383.071,Z 826.752,A -85,B 0,C 180,E1 9706.604,E2 9706.604} C_VEL
LIN {X 0,Y 378.478,Z 852.891,A -85,B 0,C 180,E1 9706.162,E2 9706.162} C_VEL
LIN {X 0,Y 373.156,Z 874.922,A -85,B 0,C 180,E1 9705.719,E2 9705.719} C_VEL
LIN {X 0,Y 365.316,Z 900.352,A -85,B 0,C 180,E1 9705.058,E2 9705.058} C_VEL
LIN {X 0,Y 357.693,Z 920.769,A -85,B 0,C 180,E1 9704.369,E2 9704.369} C_VEL
LIN {X 0,Y 347.497,Z 944.084,A -85,B 0,C 180,E1 9703.372,E2 9703.372} C_VEL
LIN {X 0,Y 337.866,Z 963.071,A -85,B 0,C 180,E1 9702.353,E2 9702.353} C_VEL
LIN {X 0,Y 326.231,Z 983.562,A -85,B 0,C 180,E1 9701.006,E2 9701.006} C_VEL
LIN {X 0,Y 313.33,Z 1003.383,A -85,B 0,C 180,E1 9699.363,E2 9699.363} C_VEL
LIN {X 0,Y 300.292,Z 1021.589,A -85,B 0,C 180,E1 9697.485,E2 9697.485} C_VEL
LIN {X 0,Y 286.341,Z 1039.034,A -85,B 0,C 180,E1 9695.218,E2 9695.218} C_VEL
LIN {X 0,Y 273.243,Z 1054.109,A -85,B 0,C 180,E1 9692.776,E2 9692.776} C_VEL
LIN {X 0,Y 257.846,Z 1070.388,A -85,B 0,C 180,E1 9689.417,E2 9689.417} C_VEL
LIN {X 0,Y 244.779,Z 1083.204,A -85,B 0,C 180,E1 9686.02,E2 9686.02} C_VEL
LIN {X 0,Y 230.253,Z 1096.636,A -85,B 0,C 180,E1 9681.413,E2 9681.413} C_VEL
LIN {X 0,Y 218.931,Z 1106.596,A -85,B 0,C 180,E1 9676.949,E2 9676.949} C_VEL
LIN {X 0,Y 207.676,Z 1116.406,A -85,B 0,C 180,E1 9671.27,E2 9671.27} C_VEL
LIN {X 0,Y 198.498,Z 1124.317,A -85,B 0,C 180,E1 9665.047,E2 9665.047} C_VEL
LIN {X 0,Y 191.348,Z 1131.009,A -85,B 0,C 180,E1 9658.054,E2 9658.054} C_VEL
LIN {X 0,Y 186.743,Z 1135.835,A -85,B 0,C 180,E1 9650.695,E2 9650.695} C_VEL
LIN {X 0,Y 184.654,Z 1138.803,A -85,B 0,C 180,E1 9644.103,E2 9644.103} C_VEL
LIN {X 0,Y 184.052,Z 1140.663,A -85,B 0,C 180,E1 9636.864,E2 9636.864} C_VEL
LIN {X 0,Y 184.124,Z 1141.006,A -85,B 0,C 180,E1 9631.245,E2 9631.245} C_VEL
LIN {X 0,Y 184.084,Z 1140.475,A -85,B 0,C 180,E1 9625.951,E2 9625.951} C_VEL
LIN {X 0,Y 184.15,Z 1138.857,A -85,B 0,C 180,E1 9619.994,E2 9619.994} C_VEL
LIN {X 0,Y 185.136,Z 1136.039,A -85,B 0,C 180,E1 9613.689,E2 9613.689} C_VEL
LIN {X 0,Y 188.054,Z 1131.438,A -85,B 0,C 180,E1 9606.498,E2 9606.498} C_VEL
LIN {X 0,Y 193.214,Z 1125.069,A -85,B 0,C 180,E1 9599.525,E2 9599.525} C_VEL
LIN {X 0,Y 199.95,Z 1117.885,A -85,B 0,C 180,E1 9593.481,E2 9593.481} C_VEL
LIN {X 0,Y 209.913,Z 1107.825,A -85,B 0,C 180,E1 9587.065,E2 9587.065} C_VEL
LIN {X 0,Y 219.927,Z 1097.842,A -85,B 0,C 180,E1 9582.177,E2 9582.177} C_VEL
LIN {X 0,Y 233.139,Z 1084.4,A -85,B 0,C 180,E1 9577.087,E2 9577.087} C_VEL
LIN {X 0,Y 245.27,Z 1071.476,A -85,B 0,C 180,E1 9573.309,E2 9573.309} C_VEL
LIN {X 0,Y 259.067,Z 1055.939,A -85,B 0,C 180,E1 9569.726,E2 9569.726} C_VEL
LIN {X 0,Y 271.879,Z 1040.299,A -85,B 0,C 180,E1 9566.895,E2 9566.895} C_VEL
LIN {X 0,Y 285.316,Z 1022.648,A -85,B 0,C 180,E1 9564.332,E2 9564.332} C_VEL
LIN {X 0,Y 297.645,Z 1004.605,A -85,B 0,C 180,E1 9562.256,E2 9562.256} C_VEL
LIN {X 0,Y 309.179,Z 986.164,A -85,B 0,C 180,E1 9560.526,E2 9560.526} C_VEL
LIN {X 0,Y 320.855,Z 965.074,A -85,B 0,C 180,E1 9558.948,E2 9558.948} C_VEL
LIN {X 0,Y 330.203,Z 946.059,A -85,B 0,C 180,E1 9557.788,E2 9557.788} C_VEL
LIN {X 0,Y 340.229,Z 922.623,A -85,B 0,C 180,E1 9556.649,E2 9556.649} C_VEL
LIN {X 0,Y 347.714,Z 902.075,A -85,B 0,C 180,E1 9555.867,E2 9555.867} C_VEL
LIN {X 0,Y 354.998,Z 878.313,A -85,B 0,C 180,E1 9555.155,E2 9555.155} C_VEL
LIN {X 0,Y 360.51,Z 855.189,A -85,B 0,C 180,E1 9554.623,E2 9554.623} C_VEL
LIN {X 0,Y 364.935,Z 830.433,A -85,B 0,C 180,E1 9554.155,E2 9554.155} C_VEL
LIN {X 0,Y 370.709,Z 776.58,A -85,B 0,C 180,E1 9553.336,E2 9553.336} C_VEL
LIN {X 0,Y 381.308,Z 672.726,A -85,B 0,C 180,E1 9551.802,E2 9551.802} C_VEL
LIN {X 0,Y 378.209,Z 666.123,A -85,B 0,C 180,E1 9549.05,E2 9549.05} C_VEL
LIN {X 0,Y 376.196,Z 661.982,A -85,B 0,C 180,E1 9546.793,E2 9546.793} C_VEL
LIN {X 0,Y 374.982,Z 659.348,A -85,B 0,C 180,E1 9545.048,E2 9545.048} C_VEL
LIN {X 0,Y 373.423,Z 655.557,A -85,B 0,C 180,E1 9541.534,E2 9541.534} C_VEL
LIN {X 0,Y 372.989,Z 655.262,A -85,B 0,C 180,E1 9536.619,E2 9536.619} C_VEL
LIN {X 0,Y 373.509,Z 655.822,A -85,B 0,C 180,E1 9534.624,E2 9534.624} C_VEL
LIN {X 0,Y 375.479,Z 660.41,A -85,B 0,C 180,E1 9530.651,E2 9530.651} C_VEL
LIN {X 0,Y 377.56,Z 664.807,A -85,B 0,C 180,E1 9528.079,E2 9528.079} C_VEL
LIN {X 0,Y 380.153,Z 670.281,A -85,B 0,C 180,E1 9525.608,E2 9525.608} C_VEL
LIN {X 0,Y 381.211,Z 672.894,A -85,B 0,C 180,E1 9524.705,E2 9524.705} C_VEL
LIN {X 0,Y 365.943,Z 819.938,A -85,B 0,C 180,E1 9522.535,E2 9522.535} C_VEL
LIN {X 0,Y 361.53,Z 846.231,A -85,B 0,C 180,E1 9522.027,E2 9522.027} C_VEL
LIN {X 0,Y 356.803,Z 866.927,A -85,B 0,C 180,E1 9521.503,E2 9521.503} C_VEL
LIN {X 0,Y 349.628,Z 891.844,A -85,B 0,C 180,E1 9520.693,E2 9520.693} C_VEL
LIN {X 0,Y 342.348,Z 912.479,A -85,B 0,C 180,E1 9519.84,E2 9519.84} C_VEL
LIN {X 0,Y 333.097,Z 935.018,A -85,B 0,C 180,E1 9518.685,E2 9518.685} C_VEL
LIN {X 0,Y 323.294,Z 955.292,A -85,B 0,C 180,E1 9517.4,E2 9517.4} C_VEL
LIN {X 0,Y 312.743,Z 974.79,A -85,B 0,C 180,E1 9515.895,E2 9515.895} C_VEL
LIN {X 0,Y 300.426,Z 994.767,A -85,B 0,C 180,E1 9513.979,E2 9513.979} C_VEL
LIN {X 0,Y 288.832,Z 1011.793,A -85,B 0,C 180,E1 9511.979,E2 9511.979} C_VEL
LIN {X 0,Y 275.384,Z 1029.616,A -85,B 0,C 180,E1 9509.376,E2 9509.376} C_VEL
LIN {X 0,Y 263.22,Z 1044.39,A -85,B 0,C 180,E1 9506.691,E2 9506.691} C_VEL
LIN {X 0,Y 249.015,Z 1060.331,A -85,B 0,C 180,E1 9503.041,E2 9503.041} C_VEL
LIN {X 0,Y 237.061,Z 1072.802,A -85,B 0,C 180,E1 9499.395,E2 9499.395} C_VEL
LIN {X 0,Y 224.465,Z 1085.344,A -85,B 0,C 180,E1 9494.734,E2 9494.734} C_VEL
LIN {X 0,Y 213.815,Z 1095.442,A -85,B 0,C 180,E1 9489.842,E2 9489.842} C_VEL
LIN {X 0,Y 203.92,Z 1104.864,A -85,B 0,C 180,E1 9483.986,E2 9483.986} C_VEL
LIN {X 0,Y 196.013,Z 1112.383,A -85,B 0,C 180,E1 9477.659,E2 9477.659} C_VEL
LIN {X 0,Y 190.229,Z 1118.446,A -85,B 0,C 180,E1 9470.942,E2 9470.942} C_VEL
LIN {X 0,Y 186.424,Z 1123.041,A -85,B 0,C 180,E1 9463.65,E2 9463.65} C_VEL
LIN {X 0,Y 184.78,Z 1125.7,A -85,B 0,C 180,E1 9457.462,E2 9457.462} C_VEL
LIN {X 0,Y 184.198,Z 1127.334,A -85,B 0,C 180,E1 9451.244,E2 9451.244} C_VEL
LIN {X 0,Y 184.143,Z 1127.967,A -85,B 0,C 180,E1 9445.016,E2 9445.016} C_VEL
LIN {X 0,Y 184.518,Z 1127.47,A -85,B 0,C 180,E1 9438.75,E2 9438.75} C_VEL
LIN {X 0,Y 185.904,Z 1125.817,A -85,B 0,C 180,E1 9432.147,E2 9432.147} C_VEL
LIN {X 0,Y 188.837,Z 1123.017,A -85,B 0,C 180,E1 9425.606,E2 9425.606} C_VEL
LIN {X 0,Y 194.948,Z 1117.782,A -85,B 0,C 180,E1 9417.763,E2 9417.763} C_VEL
LIN {X 0,Y 202.005,Z 1112.089,A -85,B 0,C 180,E1 9411.776,E2 9411.776} C_VEL
LIN {X 0,Y 212.773,Z 1103.504,A -85,B 0,C 180,E1 9405.178,E2 9405.178} C_VEL
LIN {X 0,Y 223.059,Z 1095.07,A -85,B 0,C 180,E1 9400.355,E2 9400.355} C_VEL
LIN {X 0,Y 236.26,Z 1083.89,A -85,B 0,C 180,E1 9395.437,E2 9395.437} C_VEL
LIN {X 0,Y 249.54,Z 1071.789,A -85,B 0,C 180,E1 9391.408,E2 9391.408} C_VEL
LIN {X 0,Y 263.988,Z 1057.807,A -85,B 0,C 180,E1 9387.767,E2 9387.767} C_VEL
LIN {X 0,Y 277.644,Z 1043.254,A -85,B 0,C 180,E1 9384.832,E2 9384.832} C_VEL
LIN {X 0,Y 291.644,Z 1027.165,A -85,B 0,C 180,E1 9382.228,E2 9382.228} C_VEL
LIN {X 0,Y 305.346,Z 1009.553,A -85,B 0,C 180,E1 9379.979,E2 9379.979} C_VEL
LIN {X 0,Y 318.167,Z 991.431,A -85,B 0,C 180,E1 9378.102,E2 9378.102} C_VEL
LIN {X 0,Y 330.509,Z 971.682,A -85,B 0,C 180,E1 9376.458,E2 9376.458} C_VEL
LIN {X 0,Y 340.28,Z 954.203,A -85,B 0,C 180,E1 9375.267,E2 9375.267} C_VEL
LIN {X 0,Y 350.964,Z 932.564,A -85,B 0,C 180,E1 9374.05,E2 9374.05} C_VEL
LIN {X 0,Y 359.365,Z 912.617,A -85,B 0,C 180,E1 9373.135,E2 9373.135} C_VEL
LIN {X 0,Y 367.406,Z 890.497,A -85,B 0,C 180,E1 9372.307,E2 9372.307} C_VEL
LIN {X 0,Y 374.404,Z 866.563,A -85,B 0,C 180,E1 9371.611,E2 9371.611} C_VEL
LIN {X 0,Y 379.433,Z 845.064,A -85,B 0,C 180,E1 9371.123,E2 9371.123} C_VEL
LIN {X 0,Y 383.795,Z 819.198,A -85,B 0,C 180,E1 9370.671,E2 9370.671} C_VEL
LIN {X 0,Y 398.169,Z 686.135,A -85,B 0,C 180,E1 9368.775,E2 9368.775} C_VEL
LIN {X 0,Y 396.443,Z 682.444,A -85,B 0,C 180,E1 9366.808,E2 9366.808} C_VEL
LIN {X 0,Y 395.26,Z 679.753,A -85,B 0,C 180,E1 9365.08,E2 9365.08} C_VEL
LIN {X 0,Y 393.867,Z 676.199,A -85,B 0,C 180,E1 9361.891,E2 9361.891} C_VEL
LIN {X 0,Y 393.423,Z 675.802,A -85,B 0,C 180,E1 9357.378,E2 9357.378} C_VEL
LIN {X 0,Y 394.035,Z 676.574,A -85,B 0,C 180,E1 9355.051,E2 9355.051} C_VEL
LIN {X 0,Y 395.789,Z 680.836,A -85,B 0,C 180,E1 9351.574,E2 9351.574} C_VEL
LIN {X 0,Y 397.679,Z 685.076,A -85,B 0,C 180,E1 9349.204,E2 9349.204} C_VEL
LIN {X 0,Y 398.253,Z 686.523,A -85,B 0,C 180,E1 9348.58,E2 9348.58} C_VEL
LIN {X 0,Y 394.58,Z 720.765,A -85,B 0,C 180,E1 9348.107,E2 9348.107} C_VEL
LIN {X 0,Y 393.571,Z 728.461,A -85,B 0,C 180,E1 9348.144,E2 9348.144} C_VEL
LIN {X 0,Y 390.236,Z 749.018,A -85,B 0,C 180,E1 9348.761,E2 9348.761} C_VEL
LIN {X 0,Y 389.39,Z 755.622,A -85,B 0,C 180,E1 9348.78,E2 9348.78} C_VEL
LIN {X 0,Y 381.351,Z 827.551,A -85,B 0,C 180,E1 9347.77,E2 9347.77} C_VEL
LIN {X 0,Y 376.735,Z 853.072,A -85,B 0,C 180,E1 9347.348,E2 9347.348} C_VEL
LIN {X 0,Y 371.317,Z 875.154,A -85,B 0,C 180,E1 9346.919,E2 9346.919} C_VEL
LIN {X 0,Y 363.584,Z 899.889,A -85,B 0,C 180,E1 9346.299,E2 9346.299} C_VEL
LIN {X 0,Y 355.615,Z 920.948,A -85,B 0,C 180,E1 9345.614,E2 9345.614} C_VEL
LIN {X 0,Y 345.037,Z 944.654,A -85,B 0,C 180,E1 9344.629,E2 9344.629} C_VEL
LIN {X 0,Y 335.104,Z 963.857,A -85,B 0,C 180,E1 9343.625,E2 9343.625} C_VEL
LIN {X 0,Y 322.814,Z 984.918,A -85,B 0,C 180,E1 9342.262,E2 9342.262} C_VEL
LIN {X 0,Y 310.339,Z 1003.655,A -85,B 0,C 180,E1 9340.74,E2 9340.74} C_VEL
LIN {X 0,Y 296.809,Z 1022.14,A -85,B 0,C 180,E1 9338.871,E2 9338.871} C_VEL
LIN {X 0,Y 282.202,Z 1039.865,A -85,B 0,C 180,E1 9336.59,E2 9336.59} C_VEL
LIN {X 0,Y 268.04,Z 1055.692,A -85,B 0,C 180,E1 9334.03,E2 9334.03} C_VEL
LIN {X 0,Y 253.018,Z 1070.946,A -85,B 0,C 180,E1 9330.852,E2 9330.852} C_VEL
LIN {X 0,Y 239.23,Z 1084.003,A -85,B 0,C 180,E1 9327.373,E2 9327.373} C_VEL
LIN {X 0,Y 224.558,Z 1096.969,A -85,B 0,C 180,E1 9322.848,E2 9322.848} C_VEL
LIN {X 0,Y 212.8,Z 1106.862,A -85,B 0,C 180,E1 9318.34,E2 9318.34} C_VEL
LIN {X 0,Y 200.118,Z 1117.268,A -85,B 0,C 180,E1 9312.031,E2 9312.031} C_VEL
LIN {X 0,Y 191.403,Z 1124.395,A -85,B 0,C 180,E1 9306.18,E2 9306.18} C_VEL
LIN {X 0,Y 183.72,Z 1131.086,A -85,B 0,C 180,E1 9298.807,E2 9298.807} C_VEL
LIN {X 0,Y 178.937,Z 1135.743,A -85,B 0,C 180,E1 9291.298,E2 9291.298} C_VEL
LIN {X 0,Y 176.636,Z 1138.777,A -85,B 0,C 180,E1 9284.088,E2 9284.088} C_VEL
LIN {X 0,Y 176.056,Z 1140.408,A -85,B 0,C 180,E1 9276.85,E2 9276.85} C_VEL
LIN {X 0,Y 176.131,Z 1140.696,A -85,B 0,C 180,E1 9270.976,E2 9270.976} C_VEL
LIN {X 0,Y 176.082,Z 1140.176,A -85,B 0,C 180,E1 9265.766,E2 9265.766} C_VEL
LIN {X 0,Y 176.182,Z 1138.546,A -85,B 0,C 180,E1 9259.536,E2 9259.536} C_VEL
LIN {X 0,Y 177.305,Z 1135.717,A -85,B 0,C 180,E1 9252.947,E2 9252.947} C_VEL
LIN {X 0,Y 180.716,Z 1130.868,A -85,B 0,C 180,E1 9245.149,E2 9245.149} C_VEL
LIN {X 0,Y 186.416,Z 1124.398,A -85,B 0,C 180,E1 9237.926,E2 9237.926} C_VEL
LIN {X 0,Y 194.52,Z 1116.421,A -85,B 0,C 180,E1 9231.162,E2 9231.162} C_VEL
LIN {X 0,Y 204.883,Z 1106.491,A -85,B 0,C 180,E1 9224.956,E2 9224.956} C_VEL
LIN {X 0,Y 216.127,Z 1095.854,A -85,B 0,C 180,E1 9219.827,E2 9219.827} C_VEL
LIN {X 0,Y 228.858,Z 1083.322,A -85,B 0,C 180,E1 9215.213,E2 9215.213} C_VEL
LIN {X 0,Y 240.811,Z 1071.035,A -85,B 0,C 180,E1 9211.657,E2 9211.657} C_VEL
LIN {X 0,Y 255.794,Z 1054.606,A -85,B 0,C 180,E1 9207.941,E2 9207.941} C_VEL
LIN {X 0,Y 267.857,Z 1040.281,A -85,B 0,C 180,E1 9205.395,E2 9205.395} C_VEL
LIN {X 0,Y 281.218,Z 1023.234,A -85,B 0,C 180,E1 9202.942,E2 9202.942} C_VEL
LIN {X 0,Y 294.215,Z 1004.678,A -85,B 0,C 180,E1 9200.838,E2 9200.838} C_VEL
LIN {X 0,Y 305.909,Z 986.382,A -85,B 0,C 180,E1 9199.156,E2 9199.156} C_VEL
LIN {X 0,Y 317.864,Z 965.266,A -85,B 0,C 180,E1 9197.61,E2 9197.61} C_VEL
LIN {X 0,Y 327.41,Z 946.214,A -85,B 0,C 180,E1 9196.475,E2 9196.475} C_VEL
LIN {X 0,Y 337.989,Z 921.862,A -85,B 0,C 180,E1 9195.328,E2 9195.328} C_VEL
LIN {X 0,Y 345.738,Z 900.8,A -85,B 0,C 180,E1 9194.557,E2 9194.557} C_VEL
LIN {X 0,Y 353.431,Z 875.488,A -85,B 0,C 180,E1 9193.84,E2 9193.84} C_VEL
LIN {X 0,Y 358.671,Z 853.477,A -85,B 0,C 180,E1 9193.36,E2 9193.36} C_VEL
LIN {X 0,Y 363.176,Z 827.557,A -85,B 0,C 180,E1 9192.893,E2 9192.893} C_VEL
LIN {X 0,Y 372.587,Z 739.126,A -85,B 0,C 180,E1 9191.588,E2 9191.588} C_VEL
LIN {X 0,Y 378.903,Z 678.246,A -85,B 0,C 180,E1 9190.684,E2 9190.684} C_VEL
LIN {X 0,Y 376.477,Z 672.938,A -85,B 0,C 180,E1 9188.323,E2 9188.323} C_VEL
LIN {X 0,Y 374.797,Z 669.308,A -85,B 0,C 180,E1 9186.28,E2 9186.28} C_VEL
LIN {X 0,Y 373.804,Z 667.079,A -85,B 0,C 180,E1 9184.757,E2 9184.757} C_VEL
LIN {X 0,Y 372.395,Z 663.469,A -85,B 0,C 180,E1 9181.385,E2 9181.385} C_VEL
LIN {X 0,Y 372.041,Z 663.23,A -85,B 0,C 180,E1 9176.456,E2 9176.456} C_VEL
LIN {X 0,Y 372.48,Z 663.726,A -85,B 0,C 180,E1 9174.763,E2 9174.763} C_VEL
LIN {X 0,Y 374.287,Z 668.106,A -85,B 0,C 180,E1 9170.931,E2 9170.931} C_VEL
LIN {X 0,Y 376.287,Z 672.511,A -85,B 0,C 180,E1 9168.349,E2 9168.349} C_VEL
LIN {X 0,Y 378.754,Z 677.957,A -85,B 0,C 180,E1 9165.905,E2 9165.905} C_VEL
LIN {X 0,Y 378.832,Z 678.496,A -85,B 0,C 180,E1 9165.804,E2 9165.804} C_VEL
LIN {X 0,Y 363.834,Z 820.218,A -85,B 0,C 180,E1 9163.746,E2 9163.746} C_VEL
LIN {X 0,Y 359.363,Z 846.457,A -85,B 0,C 180,E1 9163.252,E2 9163.252} C_VEL
LIN {X 0,Y 354.553,Z 867.209,A -85,B 0,C 180,E1 9162.741,E2 9162.741} C_VEL
LIN {X 0,Y 347.51,Z 891.414,A -85,B 0,C 180,E1 9161.981,E2 9161.981} C_VEL
LIN {X 0,Y 339.792,Z 912.973,A -85,B 0,C 180,E1 9161.114,E2 9161.114} C_VEL
LIN {X 0,Y 330.411,Z 935.416,A -85,B 0,C 180,E1 9159.991,E2 9159.991} C_VEL
LIN {X 0,Y 320.307,Z 955.928,A -85,B 0,C 180,E1 9158.721,E2 9158.721} C_VEL
LIN {X 0,Y 309.149,Z 976.118,A -85,B 0,C 180,E1 9157.189,E2 9157.189} C_VEL
LIN {X 0,Y 296.99,Z 995.321,A -85,B 0,C 180,E1 9155.371,E2 9155.371} C_VEL
LIN {X 0,Y 285.14,Z 1012.324,A -85,B 0,C 180,E1 9153.406,E2 9153.406} C_VEL
LIN {X 0,Y 271.364,Z 1030.108,A -85,B 0,C 180,E1 9150.841,E2 9150.841} C_VEL
LIN {X 0,Y 259.589,Z 1044.035,A -85,B 0,C 180,E1 9148.349,E2 9148.349} C_VEL
LIN {X 0,Y 245.594,Z 1059.401,A -85,B 0,C 180,E1 9144.919,E2 9144.919} C_VEL
LIN {X 0,Y 233.127,Z 1071.99,A -85,B 0,C 180,E1 9141.316,E2 9141.316} C_VEL
LIN {X 0,Y 220.478,Z 1084.195,A -85,B 0,C 180,E1 9136.899,E2 9136.899} C_VEL
LIN {X 0,Y 208.644,Z 1094.941,A -85,B 0,C 180,E1 9131.77,E2 9131.77} C_VEL
LIN {X 0,Y 198.901,Z 1103.684,A -85,B 0,C 180,E1 9126.384,E2 9126.384} C_VEL
LIN {X 0,Y 189.512,Z 1112.152,A -85,B 0,C 180,E1 9119.385,E2 9119.385} C_VEL
LIN {X 0,Y 183.528,Z 1117.902,A -85,B 0,C 180,E1 9112.965,E2 9112.965} C_VEL
LIN {X 0,Y 178.856,Z 1123.057,A -85,B 0,C 180,E1 9104.902,E2 9104.902} C_VEL
LIN {X 0,Y 176.89,Z 1125.902,A -85,B 0,C 180,E1 9098.124,E2 9098.124} C_VEL
LIN {X 0,Y 176.232,Z 1127.501,A -85,B 0,C 180,E1 9091.951,E2 9091.951} C_VEL
LIN {X 0,Y 176.132,Z 1128.16,A -85,B 0,C 180,E1 9086.094,E2 9086.094} C_VEL
LIN {X 0,Y 176.439,Z 1127.957,A -85,B 0,C 180,E1 9079.552,E2 9079.552} C_VEL
LIN {X 0,Y 177.925,Z 1126.297,A -85,B 0,C 180,E1 9071.996,E2 9071.996} C_VEL
LIN {X 0,Y 180.98,Z 1123.579,A -85,B 0,C 180,E1 9065.172,E2 9065.172} C_VEL
LIN {X 0,Y 187.076,Z 1118.76,A -85,B 0,C 180,E1 9057.328,E2 9057.328} C_VEL
LIN {X 0,Y 194.752,Z 1112.899,A -85,B 0,C 180,E1 9050.829,E2 9050.829} C_VEL
LIN {X 0,Y 204.971,Z 1105.297,A -85,B 0,C 180,E1 9044.584,E2 9044.584} C_VEL
LIN {X 0,Y 216.618,Z 1096.166,A -85,B 0,C 180,E1 9039.151,E2 9039.151} C_VEL
LIN {X 0,Y 229.289,Z 1085.942,A -85,B 0,C 180,E1 9034.492,E2 9034.492} C_VEL
LIN {X 0,Y 243.233,Z 1073.829,A -85,B 0,C 180,E1 9030.313,E2 9030.313} C_VEL
LIN {X 0,Y 256.077,Z 1061.904,A -85,B 0,C 180,E1 9027.093,E2 9027.093} C_VEL
LIN {X 0,Y 271.943,Z 1045.883,A -85,B 0,C 180,E1 9023.718,E2 9023.718} C_VEL
LIN {X 0,Y 285.389,Z 1030.943,A -85,B 0,C 180,E1 9021.257,E2 9021.257} C_VEL
LIN {X 0,Y 300.58,Z 1012.336,A -85,B 0,C 180,E1 9018.825,E2 9018.825} C_VEL
LIN {X 0,Y 312.771,Z 995.65,A -85,B 0,C 180,E1 9017.085,E2 9017.085} C_VEL
LIN {X 0,Y 325.683,Z 976.063,A -85,B 0,C 180,E1 9015.415,E2 9015.415} C_VEL
LIN {X 0,Y 337.071,Z 956.26,A -85,B 0,C 180,E1 9014.065,E2 9014.065} C_VEL
LIN {X 0,Y 347.739,Z 935.363,A -85,B 0,C 180,E1 9012.899,E2 9012.899} C_VEL
LIN {X 0,Y 357.042,Z 913.832,A -85,B 0,C 180,E1 9011.925,E2 9011.925} C_VEL
LIN {X 0,Y 364.854,Z 892.801,A -85,B 0,C 180,E1 9011.153,E2 9011.153} C_VEL
LIN {X 0,Y 372.404,Z 867.833,A -85,B 0,C 180,E1 9010.436,E2 9010.436} C_VEL
LIN {X 0,Y 377.44,Z 846.796,A -85,B 0,C 180,E1 9009.968,E2 9009.968} C_VEL
LIN {X 0,Y 382.072,Z 820.311,A -85,B 0,C 180,E1 9009.511,E2 9009.511} C_VEL
LIN {X 0,Y 396.185,Z 692.206,A -85,B 0,C 180,E1 9007.724,E2 9007.724} C_VEL
LIN {X 0,Y 394.187,Z 687.63,A -85,B 0,C 180,E1 9004.948,E2 9004.948} C_VEL
LIN {X 0,Y 392.842,Z 684.104,A -85,B 0,C 180,E1 9001.75,E2 9001.75} C_VEL
LIN {X 0,Y 392.47,Z 683.769,A -85,B 0,C 180,E1 8997.225,E2 8997.225} C_VEL
LIN {X 0,Y 393.005,Z 684.474,A -85,B 0,C 180,E1 8995.184,E2 8995.184} C_VEL
LIN {X 0,Y 394.654,Z 688.654,A -85,B 0,C 180,E1 8991.77,E2 8991.77} C_VEL
LIN {X 0,Y 396.268,Z 692.409,A -85,B 0,C 180,E1 8989.64,E2 8989.64} C_VEL
LIN {X 0,Y 389.39,Z 755.622,A -85,B 0,C 180,E1 8988.78,E2 8988.78} C_VEL
LIN {X 0,Y 388.382,Z 763.319,A -85,B 0,C 180,E1 8988.82,E2 8988.82} C_VEL
LIN {X 0,Y 385.096,Z 783.875,A -85,B 0,C 180,E1 8989.453,E2 8989.453} C_VEL
LIN {X 0,Y 384.254,Z 790.478,A -85,B 0,C 180,E1 8989.471,E2 8989.471} C_VEL
LIN {X 0,Y 379.412,Z 830.938,A -85,B 0,C 180,E1 8988.907,E2 8988.907} C_VEL
LIN {X 0,Y 374.769,Z 854.982,A -85,B 0,C 180,E1 8988.514,E2 8988.514} C_VEL
LIN {X 0,Y 368.696,Z 878.898,A -85,B 0,C 180,E1 8988.055,E2 8988.055} C_VEL
LIN {X 0,Y 361.055,Z 902.116,A -85,B 0,C 180,E1 8987.476,E2 8987.476} C_VEL
LIN {X 0,Y 352.334,Z 924.509,A -85,B 0,C 180,E1 8986.757,E2 8986.757} C_VEL
LIN {X 0,Y 341.875,Z 946.95,A -85,B 0,C 180,E1 8985.825,E2 8985.825} C_VEL
LIN {X 0,Y 331.985,Z 965.598,A -85,B 0,C 180,E1 8984.863,E2 8984.863} C_VEL
LIN {X 0,Y 318.674,Z 987.578,A -85,B 0,C 180,E1 8983.447,E2 8983.447} C_VEL
LIN {X 0,Y 306.888,Z 1004.836,A -85,B 0,C 180,E1 8982.062,E2 8982.062} C_VEL
LIN {X 0,Y 291.95,Z 1024.52,A -85,B 0,C 180,E1 8980.074,E2 8980.074} C_VEL
LIN {X 0,Y 278.229,Z 1040.696,A -85,B 0,C 180,E1 8978.002,E2 8978.002} C_VEL
LIN {X 0,Y 262.968,Z 1057.216,A -85,B 0,C 180,E1 8975.335,E2 8975.335} C_VEL
LIN {X 0,Y 248.355,Z 1071.504,A -85,B 0,C 180,E1 8972.342,E2 8972.342} C_VEL
LIN {X 0,Y 233.122,Z 1085.443,A -85,B 0,C 180,E1 8968.599,E2 8968.599} C_VEL
LIN {X 0,Y 218.369,Z 1097.825,A -85,B 0,C 180,E1 8964.142,E2 8964.142} C_VEL
LIN {X 0,Y 205.089,Z 1108.528,A -85,B 0,C 180,E1 8959.086,E2 8959.086} C_VEL
LIN {X 0,Y 192.953,Z 1117.859,A -85,B 0,C 180,E1 8953.057,E2 8953.057} C_VEL
LIN {X 0,Y 183.62,Z 1125.097,A -85,B 0,C 180,E1 8946.798,E2 8946.798} C_VEL
LIN {X 0,Y 175.577,Z 1131.595,A -85,B 0,C 180,E1 8938.951,E2 8938.951} C_VEL
LIN {X 0,Y 171.151,Z 1135.651,A -85,B 0,C 180,E1 8931.956,E2 8931.956} C_VEL
LIN {X 0,Y 168.558,Z 1138.847,A -85,B 0,C 180,E1 8923.726,E2 8923.726} C_VEL
LIN {X 0,Y 168.059,Z 1140.181,A -85,B 0,C 180,E1 8916.489,E2 8916.489} C_VEL
LIN {X 0,Y 168.138,Z 1140.385,A -85,B 0,C 180,E1 8910.681,E2 8910.681} C_VEL
LIN {X 0,Y 168.072,Z 1139.806,A -85,B 0,C 180,E1 8905.222,E2 8905.222} C_VEL
LIN {X 0,Y 168.221,Z 1138.235,A -85,B 0,C 180,E1 8899.035,E2 8899.035} C_VEL
LIN {X 0,Y 169.5,Z 1135.393,A -85,B 0,C 180,E1 8892.136,E2 8892.136} C_VEL
LIN {X 0,Y 173.069,Z 1130.765,A -85,B 0,C 180,E1 8884.322,E2 8884.322} C_VEL
LIN {X 0,Y 179.125,Z 1124.355,A -85,B 0,C 180,E1 8876.835,E2 8876.835} C_VEL
LIN {X 0,Y 186.97,Z 1117.044,A -85,B 0,C 180,E1 8870.362,E2 8870.362} C_VEL
LIN {X 0,Y 198.142,Z 1106.96,A -85,B 0,C 180,E1 8863.737,E2 8863.737} C_VEL
LIN {X 0,Y 209.158,Z 1096.994,A -85,B 0,C 180,E1 8858.774,E2 8858.774} C_VEL
LIN {X 0,Y 223.505,Z 1083.544,A -85,B 0,C 180,E1 8853.684,E2 8853.684} C_VEL
LIN {X 0,Y 235.848,Z 1071.31,A -85,B 0,C 180,E1 8850.132,E2 8850.132} C_VEL
LIN {X 0,Y 250.506,Z 1055.86,A -85,B 0,C 180,E1 8846.607,E2 8846.607} C_VEL
LIN {X 0,Y 263.627,Z 1040.738,A -85,B 0,C 180,E1 8843.925,E2 8843.925} C_VEL
LIN {X 0,Y 277.288,Z 1023.763,A -85,B 0,C 180,E1 8841.511,E2 8841.511} C_VEL
LIN {X 0,Y 290.97,Z 1004.748,A -85,B 0,C 180,E1 8839.387,E2 8839.387} C_VEL
LIN {X 0,Y 302.457,Z 987.166,A -85,B 0,C 180,E1 8837.805,E2 8837.805} C_VEL
LIN {X 0,Y 315.049,Z 965.459,A -85,B 0,C 180,E1 8836.246,E2 8836.246} C_VEL
LIN {X 0,Y 324.703,Z 946.551,A -85,B 0,C 180,E1 8835.151,E2 8835.151} C_VEL
LIN {X 0,Y 335.032,Z 923.389,A -85,B 0,C 180,E1 8834.08,E2 8834.08} C_VEL
LIN {X 0,Y 343.123,Z 901.88,A -85,B 0,C 180,E1 8833.31,E2 8833.31} C_VEL
LIN {X 0,Y 350.626,Z 878.155,A -85,B 0,C 180,E1 8832.646,E2 8832.646} C_VEL
LIN {X 0,Y 356.357,Z 854.769,A -85,B 0,C 180,E1 8832.143,E2 8832.143} C_VEL
LIN {X 0,Y 360.916,Z 830.029,A -85,B 0,C 180,E1 8831.701,E2 8831.701} C_VEL
LIN {X 0,Y 366.827,Z 776.981,A -85,B 0,C 180,E1 8830.923,E2 8830.923} C_VEL
LIN {X 0,Y 376.672,Z 683.94,A -85,B 0,C 180,E1 8829.589,E2 8829.589} C_VEL
LIN {X 0,Y 374.149,Z 678.153,A -85,B 0,C 180,E1 8826.753,E2 8826.753} C_VEL
LIN {X 0,Y 372.635,Z 674.808,A -85,B 0,C 180,E1 8824.463,E2 8824.463} C_VEL
LIN {X 0,Y 371.369,Z 671.38,A -85,B 0,C 180,E1 8821.234,E2 8821.234} C_VEL
LIN {X 0,Y 371.066,Z 671.174,A -85,B 0,C 180,E1 8816.447,E2 8816.447} C_VEL
LIN {X 0,Y 371.49,Z 671.823,A -85,B 0,C 180,E1 8814.749,E2 8814.749} C_VEL
LIN {X 0,Y 373.15,Z 675.932,A -85,B 0,C 180,E1 8811.137,E2 8811.137} C_VEL
LIN {X 0,Y 375.088,Z 680.363,A -85,B 0,C 180,E1 8808.545,E2 8808.545} C_VEL
LIN {X 0,Y 376.614,Z 683.91,A -85,B 0,C 180,E1 8806.919,E2 8806.919} C_VEL
LIN {X 0,Y 361.875,Z 820.604,A -85,B 0,C 180,E1 8804.97,E2 8804.97} C_VEL
LIN {X 0,Y 357.352,Z 846.738,A -85,B 0,C 180,E1 8804.491,E2 8804.491} C_VEL
LIN {X 0,Y 352.471,Z 867.491,A -85,B 0,C 180,E1 8803.995,E2 8803.995} C_VEL
LIN {X 0,Y 345.132,Z 892.252,A -85,B 0,C 180,E1 8803.237,E2 8803.237} C_VEL
LIN {X 0,Y 337.405,Z 913.47,A -85,B 0,C 180,E1 8802.406,E2 8802.406} C_VEL
LIN {X 0,Y 327.766,Z 936.09,A -85,B 0,C 180,E1 8801.302,E2 8801.302} C_VEL
LIN {X 0,Y 317.493,Z 956.564,A -85,B 0,C 180,E1 8800.065,E2 8800.065} C_VEL
LIN {X 0,Y 306.133,Z 976.712,A -85,B 0,C 180,E1 8798.571,E2 8798.571} C_VEL
LIN {X 0,Y 293.734,Z 995.871,A -85,B 0,C 180,E1 8796.795,E2 8796.795} C_VEL
LIN {X 0,Y 281.233,Z 1013.4,A -85,B 0,C 180,E1 8794.803,E2 8794.803} C_VEL
LIN {X 0,Y 267.527,Z 1030.6,A -85,B 0,C 180,E1 8792.35,E2 8792.35} C_VEL
LIN {X 0,Y 255.441,Z 1044.51,A -85,B 0,C 180,E1 8789.892,E2 8789.892} C_VEL
LIN {X 0,Y 241.034,Z 1059.844,A -85,B 0,C 180,E1 8786.493,E2 8786.493} C_VEL
LIN {X 0,Y 228.15,Z 1072.419,A -85,B 0,C 180,E1 8782.905,E2 8782.905} C_VEL
LIN {X 0,Y 215.014,Z 1084.612,A -85,B 0,C 180,E1 8778.479,E2 8778.479} C_VEL
LIN {X 0,Y 202.66,Z 1095.332,A -85,B 0,C 180,E1 8773.299,E2 8773.299} C_VEL
LIN {X 0,Y 192.427,Z 1104.064,A -85,B 0,C 180,E1 8767.818,E2 8767.818} C_VEL
LIN {X 0,Y 182.491,Z 1112.508,A -85,B 0,C 180,E1 8760.635,E2 8760.635} C_VEL
LIN {X 0,Y 176.207,Z 1118.151,A -85,B 0,C 180,E1 8754.115,E2 8754.115} C_VEL
LIN {X 0,Y 171.224,Z 1123.226,A -85,B 0,C 180,E1 8745.93,E2 8745.93} C_VEL
LIN {X 0,Y 169.022,Z 1126.103,A -85,B 0,C 180,E1 8738.848,E2 8738.848} C_VEL
LIN {X 0,Y 168.286,Z 1127.668,A -85,B 0,C 180,E1 8732.724,E2 8732.724} C_VEL
LIN {X 0,Y 168.133,Z 1128.356,A -85,B 0,C 180,E1 8727.273,E2 8727.273} C_VEL
LIN {X 0,Y 168.295,Z 1128.371,A -85,B 0,C 180,E1 8721.458,E2 8721.458} C_VEL
LIN {X 0,Y 169.134,Z 1127.512,A -85,B 0,C 180,E1 8714.923,E2 8714.923} C_VEL
LIN {X 0,Y 172.043,Z 1125.042,A -85,B 0,C 180,E1 8706.676,E2 8706.676} C_VEL
LIN {X 0,Y 176.884,Z 1121.323,A -85,B 0,C 180,E1 8699.419,E2 8699.419} C_VEL
LIN {X 0,Y 184.369,Z 1116.032,A -85,B 0,C 180,E1 8692.205,E2 8692.205} C_VEL
LIN {X 0,Y 194.221,Z 1108.986,A -85,B 0,C 180,E1 8685.56,E2 8685.56} C_VEL
LIN {X 0,Y 205.184,Z 1101.076,A -85,B 0,C 180,E1 8680.035,E2 8680.035} C_VEL
LIN {X 0,Y 219.484,Z 1090.19,A -85,B 0,C 180,E1 8674.455,E2 8674.455} C_VEL
LIN {X 0,Y 232.112,Z 1079.972,A -85,B 0,C 180,E1 8670.507,E2 8670.507} C_VEL
LIN {X 0,Y 247.916,Z 1066.215,A -85,B 0,C 180,E1 8666.444,E2 8666.444} C_VEL
LIN {X 0,Y 261.635,Z 1053.152,A -85,B 0,C 180,E1 8663.478,E2 8663.478} C_VEL
LIN {X 0,Y 276.786,Z 1037.492,A -85,B 0,C 180,E1 8660.668,E2 8660.668} C_VEL
LIN {X 0,Y 290.83,Z 1021.283,A -85,B 0,C 180,E1 8658.394,E2 8658.394} C_VEL
LIN {X 0,Y 304.425,Z 1004.1,A -85,B 0,C 180,E1 8656.447,E2 8656.447} C_VEL
LIN {X 0,Y 317.881,Z 984.826,A -85,B 0,C 180,E1 8654.706,E2 8654.706} C_VEL
LIN {X 0,Y 328.925,Z 967.198,A -85,B 0,C 180,E1 8653.403,E2 8653.403} C_VEL
LIN {X 0,Y 341.031,Z 945.19,A -85,B 0,C 180,E1 8652.091,E2 8652.091} C_VEL
LIN {X 0,Y 350.095,Z 926.205,A -85,B 0,C 180,E1 8651.169,E2 8651.169} C_VEL
LIN {X 0,Y 359.29,Z 904.015,A -85,B 0,C 180,E1 8650.288,E2 8650.288} C_VEL
LIN {X 0,Y 366.604,Z 882.554,A -85,B 0,C 180,E1 8649.607,E2 8649.607} C_VEL
LIN {X 0,Y 372.934,Z 860.153,A -85,B 0,C 180,E1 8649.036,E2 8649.036} C_VEL
LIN {X 0,Y 378.233,Z 835.293,A -85,B 0,C 180,E1 8648.556,E2 8648.556} C_VEL
LIN {X 0,Y 381.659,Z 812.695,A -85,B 0,C 180,E1 8648.216,E2 8648.216} C_VEL
LIN {X 0,Y 394.317,Z 698.443,A -85,B 0,C 180,E1 8646.662,E2 8646.662} C_VEL
LIN {X 0,Y 392.945,Z 695.207,A -85,B 0,C 180,E1 8644.524,E2 8644.524} C_VEL
LIN {X 0,Y 391.866,Z 692.05,A -85,B 0,C 180,E1 8641.755,E2 8641.755} C_VEL
LIN {X 0,Y 391.473,Z 691.688,A -85,B 0,C 180,E1 8637.365,E2 8637.365} C_VEL
LIN {X 0,Y 391.977,Z 692.373,A -85,B 0,C 180,E1 8635.318,E2 8635.318} C_VEL
LIN {X 0,Y 393.523,Z 696.472,A -85,B 0,C 180,E1 8631.967,E2 8631.967} C_VEL
LIN {X 0,Y 394.368,Z 698.78,A -85,B 0,C 180,E1 8630.704,E2 8630.704} C_VEL
LIN {X 0,Y 384.254,Z 790.478,A -85,B 0,C 180,E1 8629.471,E2 8629.471} C_VEL
LIN {X 0,Y 383.264,Z 798.17,A -85,B 0,C 180,E1 8629.511,E2 8629.511} C_VEL
LIN {X 0,Y 379.909,Z 818.701,A -85,B 0,C 180,E1 8630.162,E2 8630.162} C_VEL
LIN {X 0,Y 378.906,Z 825.291,A -85,B 0,C 180,E1 8630.184,E2 8630.184} C_VEL
LIN {X 0,Y 374.089,Z 851.879,A -85,B 0,C 180,E1 8629.776,E2 8629.776} C_VEL
LIN {X 0,Y 368.614,Z 873.849,A -85,B 0,C 180,E1 8629.385,E2 8629.385} C_VEL
LIN {X 0,Y 360.523,Z 899.284,A -85,B 0,C 180,E1 8628.805,E2 8628.805} C_VEL
LIN {X 0,Y 352.946,Z 918.937,A -85,B 0,C 180,E1 8628.221,E2 8628.221} C_VEL
LIN {X 0,Y 343.21,Z 940.738,A -85,B 0,C 180,E1 8627.416,E2 8627.416} C_VEL
LIN {X 0,Y 331.98,Z 962.041,A -85,B 0,C 180,E1 8626.413,E2 8626.413} C_VEL
LIN {X 0,Y 319.595,Z 982.869,A -85,B 0,C 180,E1 8625.183,E2 8625.183} C_VEL
LIN {X 0,Y 306.242,Z 1002.362,A -85,B 0,C 180,E1 8623.724,E2 8623.724} C_VEL
LIN {X 0,Y 292.717,Z 1020.224,A -85,B 0,C 180,E1 8622.051,E2 8622.051} C_VEL
LIN {X 0,Y 277.787,Z 1037.808,A -85,B 0,C 180,E1 8619.963,E2 8619.963} C_VEL
LIN {X 0,Y 263.701,Z 1052.91,A -85,B 0,C 180,E1 8617.698,E2 8617.698} C_VEL
LIN {X 0,Y 246.961,Z 1069.238,A -85,B 0,C 180,E1 8614.54,E2 8614.54} C_VEL
LIN {X 0,Y 232.568,Z 1082.075,A -85,B 0,C 180,E1 8611.291,E2 8611.291} C_VEL
LIN {X 0,Y 216.301,Z 1095.548,A -85,B 0,C 180,E1 8606.794,E2 8606.794} C_VEL
LIN {X 0,Y 202.766,Z 1105.995,A -85,B 0,C 180,E1 8602.093,E2 8602.093} C_VEL
LIN {X 0,Y 189.157,Z 1116.1,A -85,B 0,C 180,E1 8595.964,E2 8595.964} C_VEL
LIN {X 0,Y 178.719,Z 1123.619,A -85,B 0,C 180,E1 8589.628,E2 8589.628} C_VEL
LIN {X 0,Y 169.882,Z 1130.266,A -85,B 0,C 180,E1 8581.987,E2 8581.987} C_VEL
LIN {X 0,Y 163.926,Z 1135.055,A -85,B 0,C 180,E1 8573.74,E2 8573.74} C_VEL
LIN {X 0,Y 160.974,Z 1138.123,A -85,B 0,C 180,E1 8565.861,E2 8565.861} C_VEL
LIN {X 0,Y 160.047,Z 1139.843,A -85,B 0,C 180,E1 8557.539,E2 8557.539} C_VEL
LIN {X 0,Y 160.135,Z 1140.139,A -85,B 0,C 180,E1 8551.431,E2 8551.431} C_VEL
LIN {X 0,Y 160.086,Z 1139.648,A -85,B 0,C 180,E1 8545.702,E2 8545.702} C_VEL
LIN {X 0,Y 160.235,Z 1138.043,A -85,B 0,C 180,E1 8538.846,E2 8538.846} C_VEL
LIN {X 0,Y 161.616,Z 1135.237,A -85,B 0,C 180,E1 8531.607,E2 8531.607} C_VEL
LIN {X 0,Y 165.229,Z 1130.865,A -85,B 0,C 180,E1 8523.783,E2 8523.783} C_VEL
LIN {X 0,Y 171.906,Z 1124.312,A -85,B 0,C 180,E1 8515.653,E2 8515.653} C_VEL
LIN {X 0,Y 180.162,Z 1117.075,A -85,B 0,C 180,E1 8509.008,E2 8509.008} C_VEL
LIN {X 0,Y 192.383,Z 1106.652,A -85,B 0,C 180,E1 8501.993,E2 8501.993} C_VEL
LIN {X 0,Y 203.997,Z 1096.633,A -85,B 0,C 180,E1 8496.97,E2 8496.97} C_VEL
LIN {X 0,Y 219.004,Z 1083.116,A -85,B 0,C 180,E1 8491.874,E2 8491.874} C_VEL
LIN {X 0,Y 232.03,Z 1070.636,A -85,B 0,C 180,E1 8488.296,E2 8488.296} C_VEL
LIN {X 0,Y 247.679,Z 1054.526,A -85,B 0,C 180,E1 8484.723,E2 8484.723} C_VEL
LIN {X 0,Y 261.191,Z 1039.305,A -85,B 0,C 180,E1 8482.115,E2 8482.115} C_VEL
LIN {X 0,Y 275.56,Z 1021.724,A -85,B 0,C 180,E1 8479.722,E2 8479.722} C_VEL
LIN {X 0,Y 288.772,Z 1003.582,A -85,B 0,C 180,E1 8477.785,E2 8477.785} C_VEL
LIN {X 0,Y 301.37,Z 984.564,A -85,B 0,C 180,E1 8476.155,E2 8476.155} C_VEL
LIN {X 0,Y 313.306,Z 964.007,A -85,B 0,C 180,E1 8474.759,E2 8474.759} C_VEL
LIN {X 0,Y 323.167,Z 944.884,A -85,B 0,C 180,E1 8473.704,E2 8473.704} C_VEL
LIN {X 0,Y 333.604,Z 921.486,A -85,B 0,C 180,E1 8472.681,E2 8472.681} C_VEL
LIN {X 0,Y 341.4,Z 900.905,A -85,B 0,C 180,E1 8471.979,E2 8471.979} C_VEL
LIN {X 0,Y 349.114,Z 876.487,A -85,B 0,C 180,E1 8471.332,E2 8471.332} C_VEL
LIN {X 0,Y 354.692,Z 853.839,A -85,B 0,C 180,E1 8470.869,E2 8470.869} C_VEL
LIN {X 0,Y 359.285,Z 828.851,A -85,B 0,C 180,E1 8470.439,E2 8470.439} C_VEL
LIN {X 0,Y 365.852,Z 770.485,A -85,B 0,C 180,E1 8469.604,E2 8469.604} C_VEL
LIN {X 0,Y 374.556,Z 689.681,A -85,B 0,C 180,E1 8468.466,E2 8468.466} C_VEL
LIN {X 0,Y 372.534,Z 685.03,A -85,B 0,C 180,E1 8465.931,E2 8465.931} C_VEL
LIN {X 0,Y 371.477,Z 682.534,A -85,B 0,C 180,E1 8464.168,E2 8464.168} C_VEL
LIN {X 0,Y 370.346,Z 679.294,A -85,B 0,C 180,E1 8461.083,E2 8461.083} C_VEL
LIN {X 0,Y 370.092,Z 679.118,A -85,B 0,C 180,E1 8456.437,E2 8456.437} C_VEL
LIN {X 0,Y 370.463,Z 679.723,A -85,B 0,C 180,E1 8454.89,E2 8454.89} C_VEL
LIN {X 0,Y 372.017,Z 683.757,A -85,B 0,C 180,E1 8451.343,E2 8451.343} C_VEL
LIN {X 0,Y 373.893,Z 688.212,A -85,B 0,C 180,E1 8448.742,E2 8448.742} C_VEL
LIN {X 0,Y 374.486,Z 689.816,A -85,B 0,C 180,E1 8448.039,E2 8448.039} C_VEL
LIN {X 0,Y 360.099,Z 820.868,A -85,B 0,C 180,E1 8446.208,E2 8446.208} C_VEL
LIN {X 0,Y 355.509,Z 847.019,A -85,B 0,C 180,E1 8445.742,E2 8445.742} C_VEL
LIN {X 0,Y 350.54,Z 867.849,A -85,B 0,C 180,E1 8445.261,E2 8445.261} C_VEL
LIN {X 0,Y 343.109,Z 892.556,A -85,B 0,C 180,E1 8444.528,E2 8444.528} C_VEL
LIN {X 0,Y 335.388,Z 913.472,A -85,B 0,C 180,E1 8443.736,E2 8443.736} C_VEL
LIN {X 0,Y 325.646,Z 936.055,A -85,B 0,C 180,E1 8442.672,E2 8442.672} C_VEL
LIN {X 0,Y 315.29,Z 956.399,A -85,B 0,C 180,E1 8441.484,E2 8441.484} C_VEL
LIN {X 0,Y 303.721,Z 976.603,A -85,B 0,C 180,E1 8440.036,E2 8440.036} C_VEL
LIN {X 0,Y 291.08,Z 995.822,A -85,B 0,C 180,E1 8438.311,E2 8438.311} C_VEL
LIN {X 0,Y 278.552,Z 1013.052,A -85,B 0,C 180,E1 8436.411,E2 8436.411} C_VEL
LIN {X 0,Y 263.88,Z 1031.089,A -85,B 0,C 180,E1 8433.902,E2 8433.902} C_VEL
LIN {X 0,Y 250.727,Z 1045.813,A -85,B 0,C 180,E1 8431.325,E2 8431.325} C_VEL
LIN {X 0,Y 235.218,Z 1061.66,A -85,B 0,C 180,E1 8427.772,E2 8427.772} C_VEL
LIN {X 0,Y 221.963,Z 1074.129,A -85,B 0,C 180,E1 8424.153,E2 8424.153} C_VEL
LIN {X 0,Y 206.655,Z 1087.559,A -85,B 0,C 180,E1 8419.008,E2 8419.008} C_VEL
LIN {X 0,Y 195.196,Z 1097.063,A -85,B 0,C 180,E1 8414.16,E2 8414.16} C_VEL
LIN {X 0,Y 183.324,Z 1106.655,A -85,B 0,C 180,E1 8407.653,E2 8407.653} C_VEL
LIN {X 0,Y 174.485,Z 1113.745,A -85,B 0,C 180,E1 8401.048,E2 8401.048} C_VEL
LIN {X 0,Y 167.31,Z 1119.929,A -85,B 0,C 180,E1 8393.231,E2 8393.231} C_VEL
LIN {X 0,Y 162.905,Z 1124.161,A -85,B 0,C 180,E1 8385.303,E2 8385.303} C_VEL
LIN {X 0,Y 160.896,Z 1126.741,A -85,B 0,C 180,E1 8378.218,E2 8378.218} C_VEL
LIN {X 0,Y 160.212,Z 1128.365,A -85,B 0,C 180,E1 8370.715,E2 8370.715} C_VEL
LIN {X 0,Y 160.209,Z 1128.791,A -85,B 0,C 180,E1 8363.55,E2 8363.55} C_VEL
LIN {X 0,Y 160.862,Z 1128.163,A -85,B 0,C 180,E1 8356.337,E2 8356.337} C_VEL
LIN {X 0,Y 162.858,Z 1126.505,A -85,B 0,C 180,E1 8349.139,E2 8349.139} C_VEL
LIN {X 0,Y 167.612,Z 1123.165,A -85,B 0,C 180,E1 8340.714,E2 8340.714} C_VEL
LIN {X 0,Y 175.162,Z 1117.998,A -85,B 0,C 180,E1 8332.765,E2 8332.765} C_VEL
LIN {X 0,Y 184.951,Z 1111.584,A -85,B 0,C 180,E1 8325.781,E2 8325.781} C_VEL
LIN {X 0,Y 196.978,Z 1103.318,A -85,B 0,C 180,E1 8319.504,E2 8319.504} C_VEL
LIN {X 0,Y 209.678,Z 1094.287,A -85,B 0,C 180,E1 8314.413,E2 8314.413} C_VEL
LIN {X 0,Y 224.898,Z 1082.621,A -85,B 0,C 180,E1 8309.571,E2 8309.571} C_VEL
LIN {X 0,Y 238.266,Z 1071.613,A -85,B 0,C 180,E1 8306.096,E2 8306.096} C_VEL
LIN {X 0,Y 255.262,Z 1056.34,A -85,B 0,C 180,E1 8302.415,E2 8302.415} C_VEL
LIN {X 0,Y 269.011,Z 1042.725,A -85,B 0,C 180,E1 8299.884,E2 8299.884} C_VEL
LIN {X 0,Y 284.927,Z 1025.396,A -85,B 0,C 180,E1 8297.344,E2 8297.344} C_VEL
LIN {X 0,Y 298.31,Z 1009.083,A -85,B 0,C 180,E1 8295.459,E2 8295.459} C_VEL
LIN {X 0,Y 312.205,Z 990.378,A -85,B 0,C 180,E1 8293.71,E2 8293.71} C_VEL
LIN {X 0,Y 324.786,Z 970.98,A -85,B 0,C 180,E1 8292.265,E2 8292.265} C_VEL
LIN {X 0,Y 336.68,Z 950.43,A -85,B 0,C 180,E1 8291.025,E2 8291.025} C_VEL
LIN {X 0,Y 347.537,Z 928.402,A -85,B 0,C 180,E1 8289.961,E2 8289.961} C_VEL
LIN {X 0,Y 356.024,Z 908.585,A -85,B 0,C 180,E1 8289.181,E2 8289.181} C_VEL
LIN {X 0,Y 364.405,Z 885.167,A -85,B 0,C 180,E1 8288.435,E2 8288.435} C_VEL
LIN {X 0,Y 370.645,Z 863.781,A -85,B 0,C 180,E1 8287.897,E2 8287.897} C_VEL
LIN {X 0,Y 376.5,Z 837.874,A -85,B 0,C 180,E1 8287.396,E2 8287.396} C_VEL
LIN {X 0,Y 380.048,Z 815.474,A -85,B 0,C 180,E1 8287.063,E2 8287.063} C_VEL
LIN {X 0,Y 392.566,Z 704.846,A -85,B 0,C 180,E1 8285.591,E2 8285.591} C_VEL
LIN {X 0,Y 391.801,Z 702.931,A -85,B 0,C 180,E1 8284.244,E2 8284.244} C_VEL
LIN {X 0,Y 390.844,Z 699.956,A -85,B 0,C 180,E1 8281.613,E2 8281.613} C_VEL
LIN {X 0,Y 390.521,Z 699.657,A -85,B 0,C 180,E1 8277.212,E2 8277.212} C_VEL
LIN {X 0,Y 390.951,Z 700.271,A -85,B 0,C 180,E1 8275.453,E2 8275.453} C_VEL
LIN {X 0,Y 392.398,Z 704.29,A -85,B 0,C 180,E1 8272.165,E2 8272.165} C_VEL
LIN {X 0,Y 392.602,Z 705.18,A -85,B 0,C 180,E1 8271.778,E2 8271.778} C_VEL
LIN {X 0,Y 378.906,Z 825.291,A -85,B 0,C 180,E1 8270.184,E2 8270.184} C_VEL
LIN {X 0,Y 377.384,Z 834.02,A -85,B 0,C 180,E1 8270.256,E2 8270.256} C_VEL
LIN {X 0,Y 372.974,Z 852.122,A -85,B 0,C 180,E1 8270.843,E2 8270.843} C_VEL
LIN {X 0,Y 371.119,Z 859.667,A -85,B 0,C 180,E1 8270.867,E2 8270.867} C_VEL
LIN {X 0,Y 364.302,Z 883.989,A -85,B 0,C 180,E1 8270.412,E2 8270.412} C_VEL
LIN {X 0,Y 357.147,Z 904.715,A -85,B 0,C 180,E1 8269.924,E2 8269.924} C_VEL
LIN {X 0,Y 346.664,Z 929.891,A -85,B 0,C 180,E1 8269.148,E2 8269.148} C_VEL
LIN {X 0,Y 336.9,Z 949.816,A -85,B 0,C 180,E1 8268.355,E2 8268.355} C_VEL
LIN {X 0,Y 324.01,Z 972.604,A -85,B 0,C 180,E1 8267.207,E2 8267.207} C_VEL
LIN {X 0,Y 312.176,Z 990.894,A -85,B 0,C 180,E1 8266.05,E2 8266.05} C_VEL
LIN {X 0,Y 297.824,Z 1010.707,A -85,B 0,C 180,E1 8264.484,E2 8264.484} C_VEL
LIN {X 0,Y 283.74,Z 1027.92,A -85,B 0,C 180,E1 8262.746,E2 8262.746} C_VEL
LIN {X 0,Y 268.268,Z 1045.139,A -85,B 0,C 180,E1 8260.559,E2 8260.559} C_VEL
LIN {X 0,Y 252.429,Z 1060.831,A -85,B 0,C 180,E1 8257.956,E2 8257.956} C_VEL
LIN {X 0,Y 237.209,Z 1074.742,A -85,B 0,C 180,E1 8254.996,E2 8254.996} C_VEL
LIN {X 0,Y 221.236,Z 1088.021,A -85,B 0,C 180,E1 8251.259,E2 8251.259} C_VEL
LIN {X 0,Y 207.036,Z 1099.016,A -85,B 0,C 180,E1 8247.177,E2 8247.177} C_VEL
LIN {X 0,Y 190.96,Z 1110.646,A -85,B 0,C 180,E1 8241.278,E2 8241.278} C_VEL
LIN {X 0,Y 179.22,Z 1118.77,A -85,B 0,C 180,E1 8235.572,E2 8235.572} C_VEL
LIN {X 0,Y 167.319,Z 1126.889,A -85,B 0,C 180,E1 8227.557,E2 8227.557} C_VEL
LIN {X 0,Y 159.857,Z 1132.167,A -85,B 0,C 180,E1 8220.026,E2 8220.026} C_VEL
LIN {X 0,Y 154.48,Z 1136.521,A -85,B 0,C 180,E1 8210.854,E2 8210.854} C_VEL
LIN {X 0,Y 152.418,Z 1138.745,A -85,B 0,C 180,E1 8202.888,E2 8202.888} C_VEL
LIN {X 0,Y 152.062,Z 1139.699,A -85,B 0,C 180,E1 8196.039,E2 8196.039} C_VEL
LIN {X 0,Y 152.152,Z 1139.786,A -85,B 0,C 180,E1 8190.377,E2 8190.377} C_VEL
LIN {X 0,Y 152.075,Z 1139.207,A -85,B 0,C 180,E1 8184.718,E2 8184.718} C_VEL
LIN {X 0,Y 152.324,Z 1137.612,A -85,B 0,C 180,E1 8177.874,E2 8177.874} C_VEL
LIN {X 0,Y 153.87,Z 1134.914,A -85,B 0,C 180,E1 8170.645,E2 8170.645} C_VEL
LIN {X 0,Y 158.117,Z 1130.313,A -85,B 0,C 180,E1 8162.098,E2 8162.098} C_VEL
LIN {X 0,Y 165.503,Z 1123.641,A -85,B 0,C 180,E1 8153.696,E2 8153.696} C_VEL
LIN {X 0,Y 175.117,Z 1115.828,A -85,B 0,C 180,E1 8146.482,E2 8146.482} C_VEL
LIN {X 0,Y 186.915,Z 1106.26,A -85,B 0,C 180,E1 8140.095,E2 8140.095} C_VEL
LIN {X 0,Y 199.104,Z 1096.23,A -85,B 0,C 180,E1 8135.057,E2 8135.057} C_VEL
LIN {X 0,Y 214.729,Z 1082.688,A -85,B 0,C 180,E1 8129.989,E2 8129.989} C_VEL
LIN {X 0,Y 228.722,Z 1069.71,A -85,B 0,C 180,E1 8126.338,E2 8126.338} C_VEL
LIN {X 0,Y 245.128,Z 1053.19,A -85,B 0,C 180,E1 8122.799,E2 8122.799} C_VEL
LIN {X 0,Y 258.383,Z 1038.599,A -85,B 0,C 180,E1 8120.382,E2 8120.382} C_VEL
LIN {X 0,Y 273.38,Z 1020.545,A -85,B 0,C 180,E1 8118.018,E2 8118.018} C_VEL
LIN {X 0,Y 286.367,Z 1003.034,A -85,B 0,C 180,E1 8116.218,E2 8116.218} C_VEL
LIN {X 0,Y 299.641,Z 983.304,A -85,B 0,C 180,E1 8114.596,E2 8114.596} C_VEL
LIN {X 0,Y 311.324,Z 963.377,A -85,B 0,C 180,E1 8113.305,E2 8113.305} C_VEL
LIN {X 0,Y 321.335,Z 944.22,A -85,B 0,C 180,E1 8112.293,E2 8112.293} C_VEL
LIN {X 0,Y 331.916,Z 920.726,A -85,B 0,C 180,E1 8111.313,E2 8111.313} C_VEL
LIN {X 0,Y 339.809,Z 900.082,A -85,B 0,C 180,E1 8110.641,E2 8110.641} C_VEL
LIN {X 0,Y 347.827,Z 874.674,A -85,B 0,C 180,E1 8110.006,E2 8110.006} C_VEL
LIN {X 0,Y 353.264,Z 852.644,A -85,B 0,C 180,E1 8109.579,E2 8109.579} C_VEL
LIN {X 0,Y 357.942,Z 826.813,A -85,B 0,C 180,E1 8109.154,E2 8109.154} C_VEL
LIN {X 0,Y 367.499,Z 741.81,A -85,B 0,C 180,E1 8107.975,E2 8107.975} C_VEL
LIN {X 0,Y 372.544,Z 695.698,A -85,B 0,C 180,E1 8107.324,E2 8107.324} C_VEL
LIN {X 0,Y 370.915,Z 691.614,A -85,B 0,C 180,E1 8104.949,E2 8104.949} C_VEL
LIN {X 0,Y 369.371,Z 687.237,A -85,B 0,C 180,E1 8101.086,E2 8101.086} C_VEL
LIN {X 0,Y 369.118,Z 687.063,A -85,B 0,C 180,E1 8096.428,E2 8096.428} C_VEL
LIN {X 0,Y 369.44,Z 687.623,A -85,B 0,C 180,E1 8095.031,E2 8095.031} C_VEL
LIN {X 0,Y 370.89,Z 691.58,A -85,B 0,C 180,E1 8091.551,E2 8091.551} C_VEL
LIN {X 0,Y 372.515,Z 695.61,A -85,B 0,C 180,E1 8089.175,E2 8089.175} C_VEL
LIN {X 0,Y 358.47,Z 821.302,A -85,B 0,C 180,E1 8087.455,E2 8087.455} C_VEL
LIN {X 0,Y 353.844,Z 847.267,A -85,B 0,C 180,E1 8087.007,E2 8087.007} C_VEL
LIN {X 0,Y 348.816,Z 868.077,A -85,B 0,C 180,E1 8086.544,E2 8086.544} C_VEL
LIN {X 0,Y 341.334,Z 892.659,A -85,B 0,C 180,E1 8085.842,E2 8085.842} C_VEL
LIN {X 0,Y 333.694,Z 913.127,A -85,B 0,C 180,E1 8085.095,E2 8085.095} C_VEL
LIN {X 0,Y 323.894,Z 935.66,A -85,B 0,C 180,E1 8084.077,E2 8084.077} C_VEL
LIN {X 0,Y 313.329,Z 956.151,A -85,B 0,C 180,E1 8082.927,E2 8082.927} C_VEL
LIN {X 0,Y 301.942,Z 975.76,A -85,B 0,C 180,E1 8081.579,E2 8081.579} C_VEL
LIN {X 0,Y 288.634,Z 995.773,A -85,B 0,C 180,E1 8079.852,E2 8079.852} C_VEL
LIN {X 0,Y 276.009,Z 1012.818,A -85,B 0,C 180,E1 8078.035,E2 8078.035} C_VEL
LIN {X 0,Y 261.238,Z 1030.668,A -85,B 0,C 180,E1 8075.637,E2 8075.637} C_VEL
LIN {X 0,Y 247.689,Z 1045.498,A -85,B 0,C 180,E1 8073.119,E2 8073.119} C_VEL
LIN {X 0,Y 231.745,Z 1061.416,A -85,B 0,C 180,E1 8069.647,E2 8069.647} C_VEL
LIN {X 0,Y 218.057,Z 1073.899,A -85,B 0,C 180,E1 8066.096,E2 8066.096} C_VEL
LIN {X 0,Y 203.329,Z 1086.456,A -85,B 0,C 180,E1 8061.435,E2 8061.435} C_VEL
LIN {X 0,Y 190.59,Z 1096.561,A -85,B 0,C 180,E1 8056.385,E2 8056.385} C_VEL
LIN {X 0,Y 178.407,Z 1105.991,A -85,B 0,C 180,E1 8050.13,E2 8050.13} C_VEL
LIN {X 0,Y 167.969,Z 1113.807,A -85,B 0,C 180,E1 8042.8,E2 8042.8} C_VEL
LIN {X 0,Y 160.183,Z 1120.06,A -85,B 0,C 180,E1 8034.723,E2 8034.723} C_VEL
LIN {X 0,Y 155.243,Z 1124.385,A -85,B 0,C 180,E1 8026.324,E2 8026.324} C_VEL
LIN {X 0,Y 153.035,Z 1126.943,A -85,B 0,C 180,E1 8019.022,E2 8019.022} C_VEL
LIN {X 0,Y 152.228,Z 1128.532,A -85,B 0,C 180,E1 8011.506,E2 8011.506} C_VEL
LIN {X 0,Y 152.181,Z 1129.104,A -85,B 0,C 180,E1 8004.344,E2 8004.344} C_VEL
LIN {X 0,Y 152.789,Z 1128.626,A -85,B 0,C 180,E1 7996.759,E2 7996.759} C_VEL
LIN {X 0,Y 154.919,Z 1126.986,A -85,B 0,C 180,E1 7988.811,E2 7988.811} C_VEL
LIN {X 0,Y 159.123,Z 1124.198,A -85,B 0,C 180,E1 7981.063,E2 7981.063} C_VEL
LIN {X 0,Y 167.524,Z 1118.932,A -85,B 0,C 180,E1 7971.987,E2 7971.987} C_VEL
LIN {X 0,Y 176.604,Z 1113.29,A -85,B 0,C 180,E1 7965.407,E2 7965.407} C_VEL
LIN {X 0,Y 190.018,Z 1104.717,A -85,B 0,C 180,E1 7958.367,E2 7958.367} C_VEL
LIN {X 0,Y 203.1,Z 1095.836,A -85,B 0,C 180,E1 7953.182,E2 7953.182} C_VEL
LIN {X 0,Y 219.012,Z 1084.277,A -85,B 0,C 180,E1 7948.22,E2 7948.22} C_VEL
LIN {X 0,Y 233.643,Z 1072.658,A -85,B 0,C 180,E1 7944.527,E2 7944.527} C_VEL
LIN {X 0,Y 250.034,Z 1058.529,A -85,B 0,C 180,E1 7941.095,E2 7941.095} C_VEL
LIN {X 0,Y 264.635,Z 1044.514,A -85,B 0,C 180,E1 7938.49,E2 7938.49} C_VEL
LIN {X 0,Y 279.984,Z 1028.435,A -85,B 0,C 180,E1 7936.123,E2 7936.123} C_VEL
LIN {X 0,Y 294.857,Z 1010.845,A -85,B 0,C 180,E1 7934.103,E2 7934.103} C_VEL
LIN {X 0,Y 308.252,Z 993.283,A -85,B 0,C 180,E1 7932.48,E2 7932.48} C_VEL
LIN {X 0,Y 321.864,Z 973.016,A -85,B 0,C 180,E1 7930.984,E2 7930.984} C_VEL
LIN {X 0,Y 332.902,Z 954.429,A -85,B 0,C 180,E1 7929.879,E2 7929.879} C_VEL
LIN {X 0,Y 344.98,Z 930.939,A -85,B 0,C 180,E1 7928.751,E2 7928.751} C_VEL
LIN {X 0,Y 353.408,Z 911.781,A -85,B 0,C 180,E1 7928.006,E2 7928.006} C_VEL
LIN {X 0,Y 362.181,Z 888.346,A -85,B 0,C 180,E1 7927.265,E2 7927.265} C_VEL
LIN {X 0,Y 368.968,Z 865.712,A -85,B 0,C 180,E1 7926.707,E2 7926.707} C_VEL
LIN {X 0,Y 374.732,Z 841.534,A -85,B 0,C 180,E1 7926.245,E2 7926.245} C_VEL
LIN {X 0,Y 378.703,Z 817.465,A -85,B 0,C 180,E1 7925.89,E2 7925.89} C_VEL
LIN {X 0,Y 390.958,Z 711.223,A -85,B 0,C 180,E1 7924.511,E2 7924.511} C_VEL
LIN {X 0,Y 389.824,Z 707.862,A -85,B 0,C 180,E1 7921.47,E2 7921.47} C_VEL
LIN {X 0,Y 389.546,Z 707.601,A -85,B 0,C 180,E1 7917.205,E2 7917.205} C_VEL
LIN {X 0,Y 389.928,Z 708.168,A -85,B 0,C 180,E1 7915.588,E2 7915.588} C_VEL
LIN {X 0,Y 390.989,Z 711.474,A -85,B 0,C 180,E1 7912.863,E2 7912.863} C_VEL
LIN {X 0,Y 377.77,Z 825.423,A -85,B 0,C 180,E1 7911.385,E2 7911.385} C_VEL
LIN {X 0,Y 372.932,Z 851.688,A -85,B 0,C 180,E1 7910.996,E2 7910.996} C_VEL
LIN {X 0,Y 371.119,Z 859.667,A -85,B 0,C 180,E1 7910.867,E2 7910.867} C_VEL
LIN {X 0,Y 369.132,Z 867.174,A -85,B 0,C 180,E1 7910.895,E2 7910.895} C_VEL
LIN {X 0,Y 362.735,Z 885.9,A -85,B 0,C 180,E1 7911.47,E2 7911.47} C_VEL
LIN {X 0,Y 360.177,Z 893.222,A -85,B 0,C 180,E1 7911.472,E2 7911.472} C_VEL
LIN {X 0,Y 351.397,Z 916.036,A -85,B 0,C 180,E1 7910.889,E2 7910.889} C_VEL
LIN {X 0,Y 342.47,Z 935.926,A -85,B 0,C 180,E1 7910.251,E2 7910.251} C_VEL
LIN {X 0,Y 330.219,Z 959.255,A -85,B 0,C 180,E1 7909.29,E2 7909.29} C_VEL
LIN {X 0,Y 319.072,Z 977.762,A -85,B 0,C 180,E1 7908.322,E2 7908.322} C_VEL
LIN {X 0,Y 304.829,Z 998.633,A -85,B 0,C 180,E1 7906.961,E2 7906.961} C_VEL
LIN {X 0,Y 291.696,Z 1015.654,A -85,B 0,C 180,E1 7905.551,E2 7905.551} C_VEL
LIN {X 0,Y 276.574,Z 1033.421,A -85,B 0,C 180,E1 7903.711,E2 7903.711} C_VEL
LIN {X 0,Y 260.485,Z 1050.129,A -85,B 0,C 180,E1 7901.465,E2 7901.465} C_VEL
LIN {X 0,Y 244.468,Z 1065.355,A -85,B 0,C 180,E1 7898.834,E2 7898.834} C_VEL
LIN {X 0,Y 227.463,Z 1079.83,A -85,B 0,C 180,E1 7895.498,E2 7895.498} C_VEL
LIN {X 0,Y 212.114,Z 1091.907,A -85,B 0,C 180,E1 7891.825,E2 7891.825} C_VEL
LIN {X 0,Y 195.712,Z 1103.731,A -85,B 0,C 180,E1 7886.917,E2 7886.917} C_VEL
LIN {X 0,Y 181.968,Z 1113.058,A -85,B 0,C 180,E1 7881.616,E2 7881.616} C_VEL
LIN {X 0,Y 168.197,Z 1121.944,A -85,B 0,C 180,E1 7874.49,E2 7874.49} C_VEL
LIN {X 0,Y 158.768,Z 1127.961,A -85,B 0,C 180,E1 7867.654,E2 7867.654} C_VEL
LIN {X 0,Y 150.49,Z 1133.526,A -85,B 0,C 180,E1 7858.58,E2 7858.58} C_VEL
LIN {X 0,Y 146.08,Z 1136.86,A -85,B 0,C 180,E1 7850.014,E2 7850.014} C_VEL
LIN {X 0,Y 144.306,Z 1138.769,A -85,B 0,C 180,E1 7841.998,E2 7841.998} C_VEL
LIN {X 0,Y 144.078,Z 1139.552,A -85,B 0,C 180,E1 7834.378,E2 7834.378} C_VEL
LIN {X 0,Y 144.148,Z 1139.385,A -85,B 0,C 180,E1 7828.41,E2 7828.41} C_VEL
LIN {X 0,Y 144.073,Z 1138.477,A -85,B 0,C 180,E1 7822.021,E2 7822.021} C_VEL
LIN {X 0,Y 145.113,Z 1136.091,A -85,B 0,C 180,E1 7813.178,E2 7813.178} C_VEL
LIN {X 0,Y 148.681,Z 1131.92,A -85,B 0,C 180,E1 7804.079,E2 7804.079} C_VEL
LIN {X 0,Y 154.492,Z 1126.828,A -85,B 0,C 180,E1 7796.179,E2 7796.179} C_VEL
LIN {X 0,Y 164.51,Z 1118.963,A -85,B 0,C 180,E1 7787.572,E2 7787.572} C_VEL
LIN {X 0,Y 175.275,Z 1110.77,A -85,B 0,C 180,E1 7781.147,E2 7781.147} C_VEL
LIN {X 0,Y 189.814,Z 1099.526,A -85,B 0,C 180,E1 7774.738,E2 7774.738} C_VEL
LIN {X 0,Y 202.726,Z 1089.011,A -85,B 0,C 180,E1 7770.329,E2 7770.329} C_VEL
LIN {X 0,Y 218.206,Z 1075.712,A -85,B 0,C 180,E1 7766.086,E2 7766.086} C_VEL
LIN {X 0,Y 233.369,Z 1061.404,A -85,B 0,C 180,E1 7762.682,E2 7762.682} C_VEL
LIN {X 0,Y 248.69,Z 1045.825,A -85,B 0,C 180,E1 7759.808,E2 7759.808} C_VEL
LIN {X 0,Y 263.997,Z 1028.432,A -85,B 0,C 180,E1 7757.359,E2 7757.359} C_VEL
LIN {X 0,Y 277.726,Z 1011.31,A -85,B 0,C 180,E1 7755.451,E2 7755.451} C_VEL
LIN {X 0,Y 291.801,Z 991.551,A -85,B 0,C 180,E1 7753.723,E2 7753.723} C_VEL
LIN {X 0,Y 303.525,Z 973.142,A -85,B 0,C 180,E1 7752.443,E2 7752.443} C_VEL
LIN {X 0,Y 315.992,Z 950.843,A -85,B 0,C 180,E1 7751.206,E2 7751.206} C_VEL
LIN {X 0,Y 325.633,Z 930.963,A -85,B 0,C 180,E1 7750.338,E2 7750.338} C_VEL
LIN {X 0,Y 335.117,Z 908.348,A -85,B 0,C 180,E1 7749.557,E2 7749.557} C_VEL
LIN {X 0,Y 342.472,Z 887.151,A -85,B 0,C 180,E1 7748.989,E2 7748.989} C_VEL
LIN {X 0,Y 349.006,Z 864.465,A -85,B 0,C 180,E1 7748.509,E2 7748.509} C_VEL
LIN {X 0,Y 354.381,Z 839.522,A -85,B 0,C 180,E1 7748.083,E2 7748.083} C_VEL
LIN {X 0,Y 357.869,Z 816.602,A -85,B 0,C 180,E1 7747.745,E2 7747.745} C_VEL
LIN {X 0,Y 370.701,Z 701.708,A -85,B 0,C 180,E1 7746.194,E2 7746.194} C_VEL
LIN {X 0,Y 369.345,Z 698.286,A -85,B 0,C 180,E1 7743.881,E2 7743.881} C_VEL
LIN {X 0,Y 368.308,Z 695.124,A -85,B 0,C 180,E1 7740.778,E2 7740.778} C_VEL
LIN {X 0,Y 368.172,Z 695.039,A -85,B 0,C 180,E1 7736.263,E2 7736.263} C_VEL
LIN {X 0,Y 368.418,Z 695.522,A -85,B 0,C 180,E1 7735.174,E2 7735.174} C_VEL
LIN {X 0,Y 369.767,Z 699.404,A -85,B 0,C 180,E1 7731.76,E2 7731.76} C_VEL
LIN {X 0,Y 370.644,Z 701.813,A -85,B 0,C 180,E1 7730.315,E2 7730.315} C_VEL
LIN {X 0,Y 357.038,Z 821.551,A -85,B 0,C 180,E1 7728.716,E2 7728.716} C_VEL
LIN {X 0,Y 352.31,Z 847.71,A -85,B 0,C 180,E1 7728.279,E2 7728.279} C_VEL
LIN {X 0,Y 347.202,Z 868.552,A -85,B 0,C 180,E1 7727.832,E2 7727.832} C_VEL
LIN {X 0,Y 339.476,Z 893.498,A -85,B 0,C 180,E1 7727.144,E2 7727.144} C_VEL
LIN {X 0,Y 331.689,Z 914.011,A -85,B 0,C 180,E1 7726.42,E2 7726.42} C_VEL
LIN {X 0,Y 321.796,Z 936.335,A -85,B 0,C 180,E1 7725.444,E2 7725.444} C_VEL
LIN {X 0,Y 311.096,Z 956.752,A -85,B 0,C 180,E1 7724.337,E2 7724.337} C_VEL
LIN {X 0,Y 299.507,Z 976.364,A -85,B 0,C 180,E1 7723.033,E2 7723.033} C_VEL
LIN {X 0,Y 286.4,Z 995.724,A -85,B 0,C 180,E1 7721.419,E2 7721.419} C_VEL
LIN {X 0,Y 273.765,Z 1012.49,A -85,B 0,C 180,E1 7719.697,E2 7719.697} C_VEL
LIN {X 0,Y 258.015,Z 1031.157,A -85,B 0,C 180,E1 7717.269,E2 7717.269} C_VEL
LIN {X 0,Y 244.183,Z 1045.928,A -85,B 0,C 180,E1 7714.819,E2 7714.819} C_VEL
LIN {X 0,Y 227.761,Z 1061.857,A -85,B 0,C 180,E1 7711.405,E2 7711.405} C_VEL
LIN {X 0,Y 214.367,Z 1073.705,A -85,B 0,C 180,E1 7708.095,E2 7708.095} C_VEL
LIN {X 0,Y 199.038,Z 1086.356,A -85,B 0,C 180,E1 7703.493,E2 7703.493} C_VEL
LIN {X 0,Y 185.082,Z 1096.952,A -85,B 0,C 180,E1 7698.205,E2 7698.205} C_VEL
LIN {X 0,Y 172.28,Z 1106.36,A -85,B 0,C 180,E1 7691.87,E2 7691.87} C_VEL
LIN {X 0,Y 161.419,Z 1114.016,A -85,B 0,C 180,E1 7684.527,E2 7684.527} C_VEL
LIN {X 0,Y 153.166,Z 1120.168,A -85,B 0,C 180,E1 7676.354,E2 7676.354} C_VEL
LIN {X 0,Y 147.589,Z 1124.652,A -85,B 0,C 180,E1 7667.343,E2 7667.343} C_VEL
LIN {X 0,Y 145.119,Z 1127.253,A -85,B 0,C 180,E1 7659.518,E2 7659.518} C_VEL
LIN {X 0,Y 144.236,Z 1128.832,A -85,B 0,C 180,E1 7651.589,E2 7651.589} C_VEL
LIN {X 0,Y 144.181,Z 1129.37,A -85,B 0,C 180,E1 7644.428,E2 7644.428} C_VEL
LIN {X 0,Y 144.834,Z 1128.963,A -85,B 0,C 180,E1 7636.425,E2 7636.425} C_VEL
LIN {X 0,Y 147.143,Z 1127.359,A -85,B 0,C 180,E1 7628.053,E2 7628.053} C_VEL
LIN {X 0,Y 151.677,Z 1124.608,A -85,B 0,C 180,E1 7619.933,E2 7619.933} C_VEL
LIN {X 0,Y 160.641,Z 1119.423,A -85,B 0,C 180,E1 7610.519,E2 7610.519} C_VEL
LIN {X 0,Y 170.786,Z 1113.517,A -85,B 0,C 180,E1 7603.45,E2 7603.45} C_VEL
LIN {X 0,Y 184.968,Z 1104.921,A -85,B 0,C 180,E1 7596.345,E2 7596.345} C_VEL
LIN {X 0,Y 198.347,Z 1096.241,A -85,B 0,C 180,E1 7591.281,E2 7591.281} C_VEL
LIN {X 0,Y 214.461,Z 1085.011,A -85,B 0,C 180,E1 7586.469,E2 7586.469} C_VEL
LIN {X 0,Y 229.863,Z 1073.178,A -85,B 0,C 180,E1 7582.752,E2 7582.752} C_VEL
LIN {X 0,Y 246.522,Z 1059.257,A -85,B 0,C 180,E1 7579.426,E2 7579.426} C_VEL
LIN {X 0,Y 262.136,Z 1044.62,A -85,B 0,C 180,E1 7576.78,E2 7576.78} C_VEL
LIN {X 0,Y 278.255,Z 1028.052,A -85,B 0,C 180,E1 7574.434,E2 7574.434} C_VEL
LIN {X 0,Y 293.306,Z 1010.474,A -85,B 0,C 180,E1 7572.506,E2 7572.506} C_VEL
LIN {X 0,Y 307.782,Z 991.724,A -85,B 0,C 180,E1 7570.861,E2 7570.861} C_VEL
LIN {X 0,Y 320.87,Z 972.252,A -85,B 0,C 180,E1 7569.506,E2 7569.506} C_VEL
LIN {X 0,Y 332.071,Z 953.547,A -85,B 0,C 180,E1 7568.45,E2 7568.45} C_VEL
LIN {X 0,Y 343.837,Z 930.789,A -85,B 0,C 180,E1 7567.411,E2 7567.411} C_VEL
LIN {X 0,Y 352.371,Z 911.579,A -85,B 0,C 180,E1 7566.701,E2 7566.701} C_VEL
LIN {X 0,Y 361.3,Z 887.828,A -85,B 0,C 180,E1 7565.987,E2 7565.987} C_VEL
LIN {X 0,Y 367.979,Z 865.73,A -85,B 0,C 180,E1 7565.467,E2 7565.467} C_VEL
LIN {X 0,Y 373.803,Z 841.438,A -85,B 0,C 180,E1 7565.023,E2 7565.023} C_VEL
LIN {X 0,Y 377.77,Z 817.624,A -85,B 0,C 180,E1 7564.685,E2 7564.685} C_VEL
LIN {X 0,Y 389.432,Z 718.096,A -85,B 0,C 180,E1 7563.426,E2 7563.426} C_VEL
LIN {X 0,Y 388.806,Z 715.769,A -85,B 0,C 180,E1 7561.326,E2 7561.326} C_VEL
LIN {X 0,Y 388.596,Z 715.576,A -85,B 0,C 180,E1 7557.05,E2 7557.05} C_VEL
LIN {X 0,Y 388.938,Z 716.25,A -85,B 0,C 180,E1 7555.577,E2 7555.577} C_VEL
LIN {X 0,Y 389.462,Z 718.241,A -85,B 0,C 180,E1 7553.951,E2 7553.951} C_VEL
LIN {X 0,Y 376.838,Z 825.295,A -85,B 0,C 180,E1 7552.596,E2 7552.596} C_VEL
LIN {X 0,Y 371.946,Z 851.497,A -85,B 0,C 180,E1 7552.222,E2 7552.222} C_VEL
LIN {X 0,Y 366.336,Z 873.54,A -85,B 0,C 180,E1 7551.865,E2 7551.865} C_VEL
LIN {X 0,Y 360.177,Z 893.222,A -85,B 0,C 180,E1 7551.472,E2 7551.472} C_VEL
LIN {X 0,Y 357.498,Z 900.521,A -85,B 0,C 180,E1 7551.464,E2 7551.464} C_VEL
LIN {X 0,Y 349.454,Z 918.715,A -85,B 0,C 180,E1 7551.96,E2 7551.96} C_VEL
LIN {X 0,Y 346.123,Z 925.709,A -85,B 0,C 180,E1 7551.917,E2 7551.917} C_VEL
LIN {X 0,Y 335.656,Z 946.897,A -85,B 0,C 180,E1 7551.182,E2 7551.182} C_VEL
LIN {X 0,Y 324.107,Z 967.418,A -85,B 0,C 180,E1 7550.292,E2 7550.292} C_VEL
LIN {X 0,Y 310.993,Z 987.532,A -85,B 0,C 180,E1 7549.184,E2 7549.184} C_VEL
LIN {X 0,Y 298.019,Z 1005.298,A -85,B 0,C 180,E1 7547.966,E2 7547.966} C_VEL
LIN {X 0,Y 281.59,Z 1025.217,A -85,B 0,C 180,E1 7546.209,E2 7546.209} C_VEL
LIN {X 0,Y 266.804,Z 1041.232,A -85,B 0,C 180,E1 7544.398,E2 7544.398} C_VEL
LIN {X 0,Y 249.308,Z 1058.241,A -85,B 0,C 180,E1 7541.903,E2 7541.903} C_VEL
LIN {X 0,Y 234.04,Z 1071.623,A -85,B 0,C 180,E1 7539.332,E2 7539.332} C_VEL
LIN {X 0,Y 216.14,Z 1085.932,A -85,B 0,C 180,E1 7535.692,E2 7535.692} C_VEL
LIN {X 0,Y 200.759,Z 1097.076,A -85,B 0,C 180,E1 7531.831,E2 7531.831} C_VEL
LIN {X 0,Y 184.393,Z 1108.16,A -85,B 0,C 180,E1 7526.625,E2 7526.625} C_VEL
LIN {X 0,Y 169.774,Z 1117.242,A -85,B 0,C 180,E1 7520.492,E2 7520.492} C_VEL
LIN {X 0,Y 156.864,Z 1125.088,A -85,B 0,C 180,E1 7513.004,E2 7513.004} C_VEL
LIN {X 0,Y 146.82,Z 1131.019,A -85,B 0,C 180,E1 7504.42,E2 7504.42} C_VEL
LIN {X 0,Y 140.288,Z 1135.283,A -85,B 0,C 180,E1 7495.318,E2 7495.318} C_VEL
LIN {X 0,Y 136.749,Z 1138.06,A -85,B 0,C 180,E1 7485.166,E2 7485.166} C_VEL
LIN {X 0,Y 136.063,Z 1139.108,A -85,B 0,C 180,E1 7477.177,E2 7477.177} C_VEL
LIN {X 0,Y 136.158,Z 1139.229,A -85,B 0,C 180,E1 7470.842,E2 7470.842} C_VEL
LIN {X 0,Y 136.082,Z 1138.679,A -85,B 0,C 180,E1 7464.519,E2 7464.519} C_VEL
LIN {X 0,Y 136.424,Z 1137.108,A -85,B 0,C 180,E1 7456.867,E2 7456.867} C_VEL
LIN {X 0,Y 138.52,Z 1134.265,A -85,B 0,C 180,E1 7448.399,E2 7448.399} C_VEL
LIN {X 0,Y 144.033,Z 1129.391,A -85,B 0,C 180,E1 7438.624,E2 7438.624} C_VEL
LIN {X 0,Y 152.451,Z 1122.925,A -85,B 0,C 180,E1 7430.002,E2 7430.002} C_VEL
LIN {X 0,Y 163.683,Z 1114.942,A -85,B 0,C 180,E1 7422.34,E2 7422.34} C_VEL
LIN {X 0,Y 177.286,Z 1105.003,A -85,B 0,C 180,E1 7415.692,E2 7415.692} C_VEL
LIN {X 0,Y 191.744,Z 1094.141,A -85,B 0,C 180,E1 7410.386,E2 7410.386} C_VEL
LIN {X 0,Y 207.68,Z 1081.177,A -85,B 0,C 180,E1 7405.798,E2 7405.798} C_VEL
LIN {X 0,Y 222.661,Z 1068.107,A -85,B 0,C 180,E1 7402.32,E2 7402.32} C_VEL
LIN {X 0,Y 239.198,Z 1052.245,A -85,B 0,C 180,E1 7399.139,E2 7399.139} C_VEL
LIN {X 0,Y 253.771,Z 1036.896,A -85,B 0,C 180,E1 7396.773,E2 7396.773} C_VEL
LIN {X 0,Y 270.076,Z 1017.799,A -85,B 0,C 180,E1 7394.501,E2 7394.501} C_VEL
LIN {X 0,Y 283.125,Z 1000.703,A -85,B 0,C 180,E1 7392.907,E2 7392.907} C_VEL
LIN {X 0,Y 297.316,Z 979.882,A -85,B 0,C 180,E1 7391.381,E2 7391.381} C_VEL
LIN {X 0,Y 308.939,Z 960.414,A -85,B 0,C 180,E1 7390.254,E2 7390.254} C_VEL
LIN {X 0,Y 320.544,Z 938.309,A -85,B 0,C 180,E1 7389.237,E2 7389.237} C_VEL
LIN {X 0,Y 329.59,Z 918.066,A -85,B 0,C 180,E1 7388.504,E2 7388.504} C_VEL
LIN {X 0,Y 338.147,Z 895.841,A -85,B 0,C 180,E1 7387.866,E2 7387.866} C_VEL
LIN {X 0,Y 345.702,Z 871.481,A -85,B 0,C 180,E1 7387.338,E2 7387.338} C_VEL
LIN {X 0,Y 351.278,Z 848.8,A -85,B 0,C 180,E1 7386.946,E2 7386.946} C_VEL
LIN {X 0,Y 355.734,Z 823.216,A -85,B 0,C 180,E1 7386.565,E2 7386.565} C_VEL
LIN {X 0,Y 368.959,Z 708.077,A -85,B 0,C 180,E1 7385.053,E2 7385.053} C_VEL
LIN {X 0,Y 368.133,Z 705.859,A -85,B 0,C 180,E1 7383.426,E2 7383.426} C_VEL
LIN {X 0,Y 367.332,Z 703.067,A -85,B 0,C 180,E1 7380.78,E2 7380.78} C_VEL
LIN {X 0,Y 367.198,Z 702.984,A -85,B 0,C 180,E1 7376.253,E2 7376.253} C_VEL
LIN {X 0,Y 367.428,Z 703.606,A -85,B 0,C 180,E1 7375.161,E2 7375.161} C_VEL
LIN {X 0,Y 368.65,Z 707.225,A -85,B 0,C 180,E1 7371.97,E2 7371.97} C_VEL
LIN {X 0,Y 368.89,Z 708.284,A -85,B 0,C 180,E1 7371.464,E2 7371.464} C_VEL
LIN {X 0,Y 355.749,Z 822.003,A -85,B 0,C 180,E1 7369.983,E2 7369.983} C_VEL
LIN {X 0,Y 350.988,Z 847.983,A -85,B 0,C 180,E1 7369.565,E2 7369.565} C_VEL
LIN {X 0,Y 345.789,Z 868.938,A -85,B 0,C 180,E1 7369.134,E2 7369.134} C_VEL
LIN {X 0,Y 337.795,Z 894.336,A -85,B 0,C 180,E1 7368.459,E2 7368.459} C_VEL
LIN {X 0,Y 329.955,Z 914.673,A -85,B 0,C 180,E1 7367.769,E2 7367.769} C_VEL
LIN {X 0,Y 319.884,Z 937.008,A -85,B 0,C 180,E1 7366.828,E2 7366.828} C_VEL
LIN {X 0,Y 309.055,Z 957.35,A -85,B 0,C 180,E1 7365.766,E2 7365.766} C_VEL
LIN {X 0,Y 296.822,Z 977.686,A -85,B 0,C 180,E1 7364.459,E2 7364.459} C_VEL
LIN {X 0,Y 283.503,Z 996.873,A -85,B 0,C 180,E1 7362.901,E2 7362.901} C_VEL
LIN {X 0,Y 269.971,Z 1014.42,A -85,B 0,C 180,E1 7361.138,E2 7361.138} C_VEL
LIN {X 0,Y 255.007,Z 1031.646,A -85,B 0,C 180,E1 7358.941,E2 7358.941} C_VEL
LIN {X 0,Y 240.855,Z 1046.4,A -85,B 0,C 180,E1 7356.559,E2 7356.559} C_VEL
LIN {X 0,Y 223.746,Z 1062.519,A -85,B 0,C 180,E1 7353.169,E2 7353.169} C_VEL
LIN {X 0,Y 209.449,Z 1074.753,A -85,B 0,C 180,E1 7349.778,E2 7349.778} C_VEL
LIN {X 0,Y 192.935,Z 1087.762,A -85,B 0,C 180,E1 7344.969,E2 7344.969} C_VEL
LIN {X 0,Y 179.148,Z 1097.789,A -85,B 0,C 180,E1 7339.876,E2 7339.876} C_VEL
LIN {X 0,Y 165.245,Z 1107.413,A -85,B 0,C 180,E1 7333.138,E2 7333.138} C_VEL
LIN {X 0,Y 154.563,Z 1114.537,A -85,B 0,C 180,E1 7326.036,E2 7326.036} C_VEL
LIN {X 0,Y 145.649,Z 1120.73,A -85,B 0,C 180,E1 7317.385,E2 7317.385} C_VEL
LIN {X 0,Y 139.919,Z 1124.974,A -85,B 0,C 180,E1 7308.327,E2 7308.327} C_VEL
LIN {X 0,Y 137.214,Z 1127.564,A -85,B 0,C 180,E1 7300.072,E2 7300.072} C_VEL
LIN {X 0,Y 136.244,Z 1129.131,A -85,B 0,C 180,E1 7291.682,E2 7291.682} C_VEL
LIN {X 0,Y 136.198,Z 1129.661,A -85,B 0,C 180,E1 7284.101,E2 7284.101} C_VEL
LIN {X 0,Y 136.955,Z 1129.236,A -85,B 0,C 180,E1 7275.627,E2 7275.627} C_VEL
LIN {X 0,Y 139.569,Z 1127.626,A -85,B 0,C 180,E1 7266.795,E2 7266.795} C_VEL
LIN {X 0,Y 144.621,Z 1124.851,A -85,B 0,C 180,E1 7258.257,E2 7258.257} C_VEL
LIN {X 0,Y 154.255,Z 1119.698,A -85,B 0,C 180,E1 7248.611,E2 7248.611} C_VEL
LIN {X 0,Y 164.629,Z 1114.04,A -85,B 0,C 180,E1 7241.664,E2 7241.664} C_VEL
LIN {X 0,Y 178.875,Z 1105.922,A -85,B 0,C 180,E1 7234.743,E2 7234.743} C_VEL
LIN {X 0,Y 193.068,Z 1097.127,A -85,B 0,C 180,E1 7229.533,E2 7229.533} C_VEL
LIN {X 0,Y 209.351,Z 1086.313,A -85,B 0,C 180,E1 7224.842,E2 7224.842} C_VEL
LIN {X 0,Y 225.972,Z 1073.961,A -85,B 0,C 180,E1 7220.989,E2 7220.989} C_VEL
LIN {X 0,Y 242.612,Z 1060.505,A -85,B 0,C 180,E1 7217.817,E2 7217.817} C_VEL
LIN {X 0,Y 258.998,Z 1045.567,A -85,B 0,C 180,E1 7215.169,E2 7215.169} C_VEL
LIN {X 0,Y 274.071,Z 1030.456,A -85,B 0,C 180,E1 7213.069,E2 7213.069} C_VEL
LIN {X 0,Y 289.824,Z 1012.719,A -85,B 0,C 180,E1 7211.14,E2 7211.14} C_VEL
LIN {X 0,Y 303.106,Z 995.983,A -85,B 0,C 180,E1 7209.686,E2 7209.686} C_VEL
LIN {X 0,Y 318.217,Z 974.422,A -85,B 0,C 180,E1 7208.195,E2 7208.195} C_VEL
LIN {X 0,Y 329.549,Z 955.925,A -85,B 0,C 180,E1 7207.179,E2 7207.179} C_VEL
LIN {X 0,Y 341.452,Z 933.669,A -85,B 0,C 180,E1 7206.184,E2 7206.184} C_VEL
LIN {X 0,Y 350.555,Z 913.649,A -85,B 0,C 180,E1 7205.461,E2 7205.461} C_VEL
LIN {X 0,Y 359.497,Z 890.692,A -85,B 0,C 180,E1 7204.786,E2 7204.786} C_VEL
LIN {X 0,Y 366.812,Z 867.016,A -85,B 0,C 180,E1 7204.246,E2 7204.246} C_VEL
LIN {X 0,Y 372.718,Z 843.062,A -85,B 0,C 180,E1 7203.823,E2 7203.823} C_VEL
LIN {X 0,Y 376.899,Z 818.538,A -85,B 0,C 180,E1 7203.484,E2 7203.484} C_VEL
LIN {X 0,Y 388.056,Z 724.861,A -85,B 0,C 180,E1 7202.326,E2 7202.326} C_VEL
LIN {X 0,Y 387.79,Z 723.679,A -85,B 0,C 180,E1 7201.182,E2 7201.182} C_VEL
LIN {X 0,Y 387.621,Z 723.521,A -85,B 0,C 180,E1 7197.043,E2 7197.043} C_VEL
LIN {X 0,Y 387.917,Z 724.145,A -85,B 0,C 180,E1 7195.713,E2 7195.713} C_VEL
LIN {X 0,Y 388.068,Z 725.07,A -85,B 0,C 180,E1 7195.047,E2 7195.047} C_VEL
LIN {X 0,Y 376.089,Z 825.063,A -85,B 0,C 180,E1 7193.814,E2 7193.814} C_VEL
LIN {X 0,Y 371.161,Z 851.177,A -85,B 0,C 180,E1 7193.457,E2 7193.457} C_VEL
LIN {X 0,Y 365.502,Z 873.225,A -85,B 0,C 180,E1 7193.117,E2 7193.117} C_VEL
LIN {X 0,Y 357.408,Z 897.986,A -85,B 0,C 180,E1 7192.64,E2 7192.64} C_VEL
LIN {X 0,Y 349.26,Z 918.479,A -85,B 0,C 180,E1 7192.122,E2 7192.122} C_VEL
LIN {X 0,Y 346.123,Z 925.709,A -85,B 0,C 180,E1 7191.917,E2 7191.917} C_VEL
LIN {X 0,Y 342.662,Z 932.704,A -85,B 0,C 180,E1 7191.86,E2 7191.86} C_VEL
LIN {X 0,Y 333,Z 950.186,A -85,B 0,C 180,E1 7192.26,E2 7192.26} C_VEL
LIN {X 0,Y 329.098,Z 956.828,A -85,B 0,C 180,E1 7192.169,E2 7192.169} C_VEL
LIN {X 0,Y 317.618,Z 975.601,A -85,B 0,C 180,E1 7191.305,E2 7191.305} C_VEL
LIN {X 0,Y 303.884,Z 995.58,A -85,B 0,C 180,E1 7190.165,E2 7190.165} C_VEL
LIN {X 0,Y 289.453,Z 1013.87,A -85,B 0,C 180,E1 7188.831,E2 7188.831} C_VEL
LIN {X 0,Y 274.262,Z 1031.241,A -85,B 0,C 180,E1 7187.224,E2 7187.224} C_VEL
LIN {X 0,Y 257.528,Z 1048.198,A -85,B 0,C 180,E1 7185.191,E2 7185.191} C_VEL
LIN {X 0,Y 242.495,Z 1061.988,A -85,B 0,C 180,E1 7183.062,E2 7183.062} C_VEL
LIN {X 0,Y 223.556,Z 1077.648,A -85,B 0,C 180,E1 7179.855,E2 7179.855} C_VEL
LIN {X 0,Y 208.015,Z 1089.239,A -85,B 0,C 180,E1 7176.651,E2 7176.651} C_VEL
LIN {X 0,Y 190.155,Z 1101.468,A -85,B 0,C 180,E1 7172.055,E2 7172.055} C_VEL
LIN {X 0,Y 175.091,Z 1110.842,A -85,B 0,C 180,E1 7167.085,E2 7167.085} C_VEL
LIN {X 0,Y 160.361,Z 1119.552,A -85,B 0,C 180,E1 7160.64,E2 7160.64} C_VEL
LIN {X 0,Y 147.428,Z 1126.689,A -85,B 0,C 180,E1 7152.705,E2 7152.705} C_VEL
LIN {X 0,Y 137.896,Z 1132.059,A -85,B 0,C 180,E1 7143.941,E2 7143.941} C_VEL
LIN {X 0,Y 131.188,Z 1136.08,A -85,B 0,C 180,E1 7133.349,E2 7133.349} C_VEL
LIN {X 0,Y 128.598,Z 1138.068,A -85,B 0,C 180,E1 7124.407,E2 7124.407} C_VEL
LIN {X 0,Y 128.076,Z 1138.909,A -85,B 0,C 180,E1 7116.275,E2 7116.275} C_VEL
LIN {X 0,Y 128.176,Z 1138.897,A -85,B 0,C 180,E1 7110,E2 7110} C_VEL
LIN {X 0,Y 128.089,Z 1138.308,A -85,B 0,C 180,E1 7103.726,E2 7103.726} C_VEL
LIN {X 0,Y 128.587,Z 1136.676,A -85,B 0,C 180,E1 7095.592,E2 7095.592} C_VEL
LIN {X 0,Y 131.117,Z 1133.773,A -85,B 0,C 180,E1 7086.637,E2 7086.637} C_VEL
LIN {X 0,Y 137.712,Z 1128.516,A -85,B 0,C 180,E1 7076.008,E2 7076.008} C_VEL
LIN {X 0,Y 146.656,Z 1122.252,A -85,B 0,C 180,E1 7067.547,E2 7067.547} C_VEL
LIN {X 0,Y 158.777,Z 1114.183,A -85,B 0,C 180,E1 7059.799,E2 7059.799} C_VEL
LIN {X 0,Y 172.839,Z 1104.416,A -85,B 0,C 180,E1 7053.339,E2 7053.339} C_VEL
LIN {X 0,Y 188.097,Z 1093.431,A -85,B 0,C 180,E1 7048.063,E2 7048.063} C_VEL
LIN {X 0,Y 204.404,Z 1080.579,A -85,B 0,C 180,E1 7043.648,E2 7043.648} C_VEL
LIN {X 0,Y 220.393,Z 1067.02,A -85,B 0,C 180,E1 7040.17,E2 7040.17} C_VEL
LIN {X 0,Y 237.065,Z 1051.324,A -85,B 0,C 180,E1 7037.172,E2 7037.172} C_VEL
LIN {X 0,Y 251.514,Z 1036.408,A -85,B 0,C 180,E1 7034.973,E2 7034.973} C_VEL
LIN {X 0,Y 268.182,Z 1017.214,A -85,B 0,C 180,E1 7032.792,E2 7032.792} C_VEL
LIN {X 0,Y 281.524,Z 999.997,A -85,B 0,C 180,E1 7031.265,E2 7031.265} C_VEL
LIN {X 0,Y 296.277,Z 978.539,A -85,B 0,C 180,E1 7029.782,E2 7029.782} C_VEL
LIN {X 0,Y 307.556,Z 959.843,A -85,B 0,C 180,E1 7028.759,E2 7028.759} C_VEL
LIN {X 0,Y 318.938,Z 938.45,A -85,B 0,C 180,E1 7027.827,E2 7027.827} C_VEL
LIN {X 0,Y 328.488,Z 917.298,A -85,B 0,C 180,E1 7027.104,E2 7027.104} C_VEL
LIN {X 0,Y 337.134,Z 895.009,A -85,B 0,C 180,E1 7026.503,E2 7026.503} C_VEL
LIN {X 0,Y 344.641,Z 870.896,A -85,B 0,C 180,E1 7026.012,E2 7026.012} C_VEL
LIN {X 0,Y 350.344,Z 847.832,A -85,B 0,C 180,E1 7025.635,E2 7025.635} C_VEL
LIN {X 0,Y 354.747,Z 822.55,A -85,B 0,C 180,E1 7025.275,E2 7025.275} C_VEL
LIN {X 0,Y 367.369,Z 714.403,A -85,B 0,C 180,E1 7023.902,E2 7023.902} C_VEL
LIN {X 0,Y 366.316,Z 710.985,A -85,B 0,C 180,E1 7020.626,E2 7020.626} C_VEL
LIN {X 0,Y 366.224,Z 710.929,A -85,B 0,C 180,E1 7016.243,E2 7016.243} C_VEL
LIN {X 0,Y 366.409,Z 711.503,A -85,B 0,C 180,E1 7015.304,E2 7015.304} C_VEL
LIN {X 0,Y 367.327,Z 714.395,A -85,B 0,C 180,E1 7012.628,E2 7012.628} C_VEL
LIN {X 0,Y 354.653,Z 822.318,A -85,B 0,C 180,E1 7011.26,E2 7011.26} C_VEL
LIN {X 0,Y 349.843,Z 848.247,A -85,B 0,C 180,E1 7010.86,E2 7010.86} C_VEL
LIN {X 0,Y 344.585,Z 869.206,A -85,B 0,C 180,E1 7010.449,E2 7010.449} C_VEL
LIN {X 0,Y 336.762,Z 893.895,A -85,B 0,C 180,E1 7009.825,E2 7009.825} C_VEL
LIN {X 0,Y 328.496,Z 915.115,A -85,B 0,C 180,E1 7009.139,E2 7009.139} C_VEL
LIN {X 0,Y 318.16,Z 937.68,A -85,B 0,C 180,E1 7008.227,E2 7008.227} C_VEL
LIN {X 0,Y 307.556,Z 957.342,A -85,B 0,C 180,E1 7007.247,E2 7007.247} C_VEL
LIN {X 0,Y 295.23,Z 977.571,A -85,B 0,C 180,E1 7006.008,E2 7006.008} C_VEL
LIN {X 0,Y 281.694,Z 996.824,A -85,B 0,C 180,E1 7004.517,E2 7004.517} C_VEL
LIN {X 0,Y 268.297,Z 1013.93,A -85,B 0,C 180,E1 7002.877,E2 7002.877} C_VEL
LIN {X 0,Y 252.221,Z 1032.134,A -85,B 0,C 180,E1 7000.651,E2 7000.651} C_VEL
LIN {X 0,Y 237.757,Z 1046.872,A -85,B 0,C 180,E1 6998.345,E2 6998.345} C_VEL
LIN {X 0,Y 220.468,Z 1062.739,A -85,B 0,C 180,E1 6995.103,E2 6995.103} C_VEL
LIN {X 0,Y 206.258,Z 1074.559,A -85,B 0,C 180,E1 6991.921,E2 6991.921} C_VEL
LIN {X 0,Y 189.833,Z 1087.159,A -85,B 0,C 180,E1 6987.432,E2 6987.432} C_VEL
LIN {X 0,Y 175.029,Z 1097.491,A -85,B 0,C 180,E1 6982.319,E2 6982.319} C_VEL
LIN {X 0,Y 160.74,Z 1106.985,A -85,B 0,C 180,E1 6975.837,E2 6975.837} C_VEL
LIN {X 0,Y 148.578,Z 1114.581,A -85,B 0,C 180,E1 6968.253,E2 6968.253} C_VEL
LIN {X 0,Y 138.857,Z 1120.853,A -85,B 0,C 180,E1 6959.318,E2 6959.318} C_VEL
LIN {X 0,Y 132.295,Z 1125.296,A -85,B 0,C 180,E1 6949.424,E2 6949.424} C_VEL
LIN {X 0,Y 129.323,Z 1127.874,A -85,B 0,C 180,E1 6940.694,E2 6940.694} C_VEL
LIN {X 0,Y 128.24,Z 1129.497,A -85,B 0,C 180,E1 6931.34,E2 6931.34} C_VEL
LIN {X 0,Y 128.236,Z 1129.969,A -85,B 0,C 180,E1 6923.283,E2 6923.283} C_VEL
LIN {X 0,Y 129.273,Z 1129.385,A -85,B 0,C 180,E1 6913.832,E2 6913.832} C_VEL
LIN {X 0,Y 132.269,Z 1127.785,A -85,B 0,C 180,E1 6904.955,E2 6904.955} C_VEL
LIN {X 0,Y 138.311,Z 1124.819,A -85,B 0,C 180,E1 6895.675,E2 6895.675} C_VEL
LIN {X 0,Y 148.607,Z 1119.69,A -85,B 0,C 180,E1 6886.13,E2 6886.13} C_VEL
LIN {X 0,Y 159.795,Z 1113.973,A -85,B 0,C 180,E1 6879.112,E2 6879.112} C_VEL
LIN {X 0,Y 175.615,Z 1105.331,A -85,B 0,C 180,E1 6871.967,E2 6871.967} C_VEL
LIN {X 0,Y 189.846,Z 1096.867,A -85,B 0,C 180,E1 6867.114,E2 6867.114} C_VEL
LIN {X 0,Y 207.591,Z 1085.346,A -85,B 0,C 180,E1 6862.362,E2 6862.362} C_VEL
LIN {X 0,Y 223.138,Z 1074.114,A -85,B 0,C 180,E1 6859.003,E2 6859.003} C_VEL
LIN {X 0,Y 240.211,Z 1060.641,A -85,B 0,C 180,E1 6855.939,E2 6855.939} C_VEL
LIN {X 0,Y 256.963,Z 1045.672,A -85,B 0,C 180,E1 6853.394,E2 6853.394} C_VEL
LIN {X 0,Y 272.33,Z 1030.543,A -85,B 0,C 180,E1 6851.384,E2 6851.384} C_VEL
LIN {X 0,Y 288.451,Z 1012.647,A -85,B 0,C 180,E1 6849.53,E2 6849.53} C_VEL
LIN {X 0,Y 302.01,Z 995.786,A -85,B 0,C 180,E1 6848.138,E2 6848.138} C_VEL
LIN {X 0,Y 317.157,Z 974.394,A -85,B 0,C 180,E1 6846.736,E2 6846.736} C_VEL
LIN {X 0,Y 328.75,Z 955.662,A -85,B 0,C 180,E1 6845.76,E2 6845.76} C_VEL
LIN {X 0,Y 341.154,Z 932.515,A -85,B 0,C 180,E1 6844.786,E2 6844.786} C_VEL
LIN {X 0,Y 349.877,Z 913.45,A -85,B 0,C 180,E1 6844.14,E2 6844.14} C_VEL
LIN {X 0,Y 358.858,Z 890.524,A -85,B 0,C 180,E1 6843.503,E2 6843.503} C_VEL
LIN {X 0,Y 366.149,Z 867.1,A -85,B 0,C 180,E1 6842.994,E2 6842.994} C_VEL
LIN {X 0,Y 372.141,Z 842.935,A -85,B 0,C 180,E1 6842.589,E2 6842.589} C_VEL
LIN {X 0,Y 376.333,Z 818.475,A -85,B 0,C 180,E1 6842.266,E2 6842.266} C_VEL
LIN {X 0,Y 386.825,Z 731.633,A -85,B 0,C 180,E1 6841.226,E2 6841.226} C_VEL
LIN {X 0,Y 386.647,Z 731.467,A -85,B 0,C 180,E1 6837.035,E2 6837.035} C_VEL
LIN {X 0,Y 386.818,Z 731.904,A -85,B 0,C 180,E1 6836.15,E2 6836.15} C_VEL
LIN {X 0,Y 375.495,Z 824.935,A -85,B 0,C 180,E1 6835.034,E2 6835.034} C_VEL
LIN {X 0,Y 370.518,Z 850.987,A -85,B 0,C 180,E1 6834.694,E2 6834.694} C_VEL
LIN {X 0,Y 364.813,Z 873.018,A -85,B 0,C 180,E1 6834.374,E2 6834.374} C_VEL
LIN {X 0,Y 356.471,Z 898.239,A -85,B 0,C 180,E1 6833.916,E2 6833.916} C_VEL
LIN {X 0,Y 348.251,Z 918.667,A -85,B 0,C 180,E1 6833.43,E2 6833.43} C_VEL
LIN {X 0,Y 337.18,Z 941.994,A -85,B 0,C 180,E1 6832.724,E2 6832.724} C_VEL
LIN {X 0,Y 329.098,Z 956.828,A -85,B 0,C 180,E1 6832.169,E2 6832.169} C_VEL
LIN {X 0,Y 325.033,Z 963.517,A -85,B 0,C 180,E1 6832.063,E2 6832.063} C_VEL
LIN {X 0,Y 313.745,Z 980.039,A -85,B 0,C 180,E1 6832.361,E2 6832.361} C_VEL
LIN {X 0,Y 309.256,Z 986.268,A -85,B 0,C 180,E1 6832.212,E2 6832.212} C_VEL
LIN {X 0,Y 296.006,Z 1004.015,A -85,B 0,C 180,E1 6831.134,E2 6831.134} C_VEL
LIN {X 0,Y 279.086,Z 1024.048,A -85,B 0,C 180,E1 6829.566,E2 6829.566} C_VEL
LIN {X 0,Y 264.225,Z 1039.677,A -85,B 0,C 180,E1 6827.987,E2 6827.987} C_VEL
LIN {X 0,Y 246.505,Z 1056.428,A -85,B 0,C 180,E1 6825.802,E2 6825.802} C_VEL
LIN {X 0,Y 230.5,Z 1069.918,A -85,B 0,C 180,E1 6823.473,E2 6823.473} C_VEL
LIN {X 0,Y 213.255,Z 1083.196,A -85,B 0,C 180,E1 6820.465,E2 6820.465} C_VEL
LIN {X 0,Y 195.094,Z 1095.659,A -85,B 0,C 180,E1 6816.551,E2 6816.551} C_VEL
LIN {X 0,Y 178.784,Z 1105.935,A -85,B 0,C 180,E1 6812.087,E2 6812.087} C_VEL
LIN {X 0,Y 161.723,Z 1115.716,A -85,B 0,C 180,E1 6805.944,E2 6805.944} C_VEL
LIN {X 0,Y 148.568,Z 1122.771,A -85,B 0,C 180,E1 6799.51,E2 6799.51} C_VEL
LIN {X 0,Y 135.229,Z 1129.656,A -85,B 0,C 180,E1 6790.037,E2 6790.037} C_VEL
LIN {X 0,Y 127.043,Z 1133.923,A -85,B 0,C 180,E1 6780.769,E2 6780.769} C_VEL
LIN {X 0,Y 121.751,Z 1137.113,A -85,B 0,C 180,E1 6769.677,E2 6769.677} C_VEL
LIN {X 0,Y 120.107,Z 1138.486,A -85,B 0,C 180,E1 6759.101,E2 6759.101} C_VEL
LIN {X 0,Y 120.145,Z 1138.692,A -85,B 0,C 180,E1 6751.908,E2 6751.908} C_VEL
LIN {X 0,Y 120.101,Z 1138.363,A -85,B 0,C 180,E1 6745.703,E2 6745.703} C_VEL
LIN {X 0,Y 120.441,Z 1136.843,A -85,B 0,C 180,E1 6736.558,E2 6736.558} C_VEL
LIN {X 0,Y 123.022,Z 1133.952,A -85,B 0,C 180,E1 6726.53,E2 6726.53} C_VEL
LIN {X 0,Y 128.81,Z 1129.616,A -85,B 0,C 180,E1 6716.555,E2 6716.555} C_VEL
LIN {X 0,Y 139.153,Z 1122.836,A -85,B 0,C 180,E1 6706.385,E2 6706.385} C_VEL
LIN {X 0,Y 150.557,Z 1115.662,A -85,B 0,C 180,E1 6699.01,E2 6699.01} C_VEL
LIN {X 0,Y 166.028,Z 1105.632,A -85,B 0,C 180,E1 6691.879,E2 6691.879} C_VEL
LIN {X 0,Y 180.519,Z 1095.668,A -85,B 0,C 180,E1 6686.902,E2 6686.902} C_VEL
LIN {X 0,Y 197.75,Z 1082.917,A -85,B 0,C 180,E1 6682.284,E2 6682.284} C_VEL
LIN {X 0,Y 214.037,Z 1069.631,A -85,B 0,C 180,E1 6678.805,E2 6678.805} C_VEL
LIN {X 0,Y 231.649,Z 1053.885,A -85,B 0,C 180,E1 6675.728,E2 6675.728} C_VEL
LIN {X 0,Y 246.797,Z 1038.747,A -85,B 0,C 180,E1 6673.503,E2 6673.503} C_VEL
LIN {X 0,Y 262.721,Z 1021.269,A -85,B 0,C 180,E1 6671.501,E2 6671.501} C_VEL
LIN {X 0,Y 277.577,Z 1002.696,A -85,B 0,C 180,E1 6669.867,E2 6669.867} C_VEL
LIN {X 0,Y 291.212,Z 983.737,A -85,B 0,C 180,E1 6668.557,E2 6668.557} C_VEL
LIN {X 0,Y 304.509,Z 962.495,A -85,B 0,C 180,E1 6667.407,E2 6667.407} C_VEL
LIN {X 0,Y 315.046,Z 943.372,A -85,B 0,C 180,E1 6666.585,E2 6666.585} C_VEL
LIN {X 0,Y 326.083,Z 920.072,A -85,B 0,C 180,E1 6665.795,E2 6665.795} C_VEL
LIN {X 0,Y 334.367,Z 899.364,A -85,B 0,C 180,E1 6665.249,E2 6665.249} C_VEL
LIN {X 0,Y 342.597,Z 874.512,A -85,B 0,C 180,E1 6664.749,E2 6664.749} C_VEL
LIN {X 0,Y 348.382,Z 852.112,A -85,B 0,C 180,E1 6664.396,E2 6664.396} C_VEL
LIN {X 0,Y 353.251,Z 826.864,A -85,B 0,C 180,E1 6664.042,E2 6664.042} C_VEL
LIN {X 0,Y 360.968,Z 763.15,A -85,B 0,C 180,E1 6663.247,E2 6663.247} C_VEL
LIN {X 0,Y 365.855,Z 721.186,A -85,B 0,C 180,E1 6662.706,E2 6662.706} C_VEL
LIN {X 0,Y 365.303,Z 718.905,A -85,B 0,C 180,E1 6660.47,E2 6660.47} C_VEL
LIN {X 0,Y 365.249,Z 718.875,A -85,B 0,C 180,E1 6656.233,E2 6656.233} C_VEL
LIN {X 0,Y 365.485,Z 719.932,A -85,B 0,C 180,E1 6654.978,E2 6654.978} C_VEL
LIN {X 0,Y 365.816,Z 721.363,A -85,B 0,C 180,E1 6653.79,E2 6653.79} C_VEL
LIN {X 0,Y 353.722,Z 822.726,A -85,B 0,C 180,E1 6652.544,E2 6652.544} C_VEL
LIN {X 0,Y 348.849,Z 848.64,A -85,B 0,C 180,E1 6652.161,E2 6652.161} C_VEL
LIN {X 0,Y 343.504,Z 869.688,A -85,B 0,C 180,E1 6651.768,E2 6651.768} C_VEL
LIN {X 0,Y 335.267,Z 895.206,A -85,B 0,C 180,E1 6651.149,E2 6651.149} C_VEL
LIN {X 0,Y 327.148,Z 915.737,A -85,B 0,C 180,E1 6650.514,E2 6650.514} C_VEL
LIN {X 0,Y 316.395,Z 938.786,A -85,B 0,C 180,E1 6649.622,E2 6649.622} C_VEL
LIN {X 0,Y 305.556,Z 958.549,A -85,B 0,C 180,E1 6648.677,E2 6648.677} C_VEL
LIN {X 0,Y 292.936,Z 978.853,A -85,B 0,C 180,E1 6647.48,E2 6647.48} C_VEL
LIN {X 0,Y 279.203,Z 997.974,A -85,B 0,C 180,E1 6646.053,E2 6646.053} C_VEL
LIN {X 0,Y 264.759,Z 1016.021,A -85,B 0,C 180,E1 6644.374,E2 6644.374} C_VEL
LIN {X 0,Y 248.787,Z 1033.532,A -85,B 0,C 180,E1 6642.274,E2 6642.274} C_VEL
LIN {X 0,Y 233.186,Z 1049.002,A -85,B 0,C 180,E1 6639.895,E2 6639.895} C_VEL
LIN {X 0,Y 216.244,Z 1063.961,A -85,B 0,C 180,E1 6636.857,E2 6636.857} C_VEL
LIN {X 0,Y 200.985,Z 1076.229,A -85,B 0,C 180,E1 6633.572,E2 6633.572} C_VEL
LIN {X 0,Y 183.357,Z 1089.067,A -85,B 0,C 180,E1 6628.888,E2 6628.888} C_VEL
LIN {X 0,Y 169.137,Z 1098.567,A -85,B 0,C 180,E1 6624.087,E2 6624.087} C_VEL
LIN {X 0,Y 153.206,Z 1108.489,A -85,B 0,C 180,E1 6616.968,E2 6616.968} C_VEL
LIN {X 0,Y 141.801,Z 1115.229,A -85,B 0,C 180,E1 6609.917,E2 6609.917} C_VEL
LIN {X 0,Y 131.495,Z 1121.397,A -85,B 0,C 180,E1 6600.629,E2 6600.629} C_VEL
LIN {X 0,Y 124.725,Z 1125.618,A -85,B 0,C 180,E1 6590.655,E2 6590.655} C_VEL
LIN {X 0,Y 121.447,Z 1128.185,A -85,B 0,C 180,E1 6581.396,E2 6581.396} C_VEL
LIN {X 0,Y 120.247,Z 1129.796,A -85,B 0,C 180,E1 6571.429,E2 6571.429} C_VEL
LIN {X 0,Y 120.253,Z 1130.254,A -85,B 0,C 180,E1 6562.835,E2 6562.835} C_VEL
LIN {X 0,Y 121.494,Z 1129.649,A -85,B 0,C 180,E1 6552.685,E2 6552.685} C_VEL
LIN {X 0,Y 124.877,Z 1128.052,A -85,B 0,C 180,E1 6543.359,E2 6543.359} C_VEL
LIN {X 0,Y 131.947,Z 1124.925,A -85,B 0,C 180,E1 6533.226,E2 6533.226} C_VEL
LIN {X 0,Y 142.741,Z 1119.928,A -85,B 0,C 180,E1 6523.821,E2 6523.821} C_VEL
LIN {X 0,Y 154.682,Z 1114.201,A -85,B 0,C 180,E1 6516.72,E2 6516.72} C_VEL
LIN {X 0,Y 171.354,Z 1105.536,A -85,B 0,C 180,E1 6509.605,E2 6509.605} C_VEL
LIN {X 0,Y 186.976,Z 1096.608,A -85,B 0,C 180,E1 6504.617,E2 6504.617} C_VEL
LIN {X 0,Y 206.29,Z 1084.336,A -85,B 0,C 180,E1 6499.834,E2 6499.834} C_VEL
LIN {X 0,Y 222.303,Z 1073.008,A -85,B 0,C 180,E1 6496.654,E2 6496.654} C_VEL
LIN {X 0,Y 241.634,Z 1057.718,A -85,B 0,C 180,E1 6493.482,E2 6493.482} C_VEL
LIN {X 0,Y 257.004,Z 1044.094,A -85,B 0,C 180,E1 6491.354,E2 6491.354} C_VEL
LIN {X 0,Y 274.547,Z 1026.748,A -85,B 0,C 180,E1 6489.257,E2 6489.257} C_VEL
LIN {X 0,Y 288.77,Z 1010.863,A -85,B 0,C 180,E1 6487.761,E2 6487.761} C_VEL
LIN {X 0,Y 303.829,Z 992.152,A -85,B 0,C 180,E1 6486.344,E2 6486.344} C_VEL
LIN {X 0,Y 317.66,Z 972.296,A -85,B 0,C 180,E1 6485.159,E2 6485.159} C_VEL
LIN {X 0,Y 330.493,Z 951.482,A -85,B 0,C 180,E1 6484.164,E2 6484.164} C_VEL
LIN {X 0,Y 342.038,Z 929.344,A -85,B 0,C 180,E1 6483.318,E2 6483.318} C_VEL
LIN {X 0,Y 351.84,Z 907.577,A -85,B 0,C 180,E1 6482.651,E2 6482.651} C_VEL
LIN {X 0,Y 360.204,Z 884.891,A -85,B 0,C 180,E1 6482.097,E2 6482.097} C_VEL
LIN {X 0,Y 366.79,Z 863.202,A -85,B 0,C 180,E1 6481.669,E2 6481.669} C_VEL
LIN {X 0,Y 372.711,Z 837.62,A -85,B 0,C 180,E1 6481.282,E2 6481.282} C_VEL
LIN {X 0,Y 376.379,Z 815.329,A -85,B 0,C 180,E1 6481.009,E2 6481.009} C_VEL
LIN {X 0,Y 385.621,Z 739.352,A -85,B 0,C 180,E1 6480.111,E2 6480.111} C_VEL
LIN {X 0,Y 385.619,Z 739.503,A -85,B 0,C 180,E1 6477.252,E2 6477.252} C_VEL
LIN {X 0,Y 375.058,Z 824.915,A -85,B 0,C 180,E1 6476.257,E2 6476.257} C_VEL
LIN {X 0,Y 370.049,Z 850.796,A -85,B 0,C 180,E1 6475.935,E2 6475.935} C_VEL
LIN {X 0,Y 364.27,Z 872.919,A -85,B 0,C 180,E1 6475.633,E2 6475.633} C_VEL
LIN {X 0,Y 356.201,Z 897.21,A -85,B 0,C 180,E1 6475.222,E2 6475.222} C_VEL
LIN {X 0,Y 347.911,Z 917.727,A -85,B 0,C 180,E1 6474.772,E2 6474.772} C_VEL
LIN {X 0,Y 337.224,Z 940.287,A -85,B 0,C 180,E1 6474.145,E2 6474.145} C_VEL
LIN {X 0,Y 325.552,Z 961.161,A -85,B 0,C 180,E1 6473.395,E2 6473.395} C_VEL
LIN {X 0,Y 312.188,Z 982.173,A -85,B 0,C 180,E1 6472.432,E2 6472.432} C_VEL
LIN {X 0,Y 309.256,Z 986.268,A -85,B 0,C 180,E1 6472.212,E2 6472.212} C_VEL
LIN {X 0,Y 304.632,Z 992.574,A -85,B 0,C 180,E1 6472.048,E2 6472.048} C_VEL
LIN {X 0,Y 291.787,Z 1008.043,A -85,B 0,C 180,E1 6472.239,E2 6472.239} C_VEL
LIN {X 0,Y 286.778,Z 1013.72,A -85,B 0,C 180,E1 6472.028,E2 6472.028} C_VEL
LIN {X 0,Y 270.648,Z 1031.599,A -85,B 0,C 180,E1 6470.546,E2 6470.546} C_VEL
LIN {X 0,Y 253.833,Z 1047.973,A -85,B 0,C 180,E1 6468.771,E2 6468.771} C_VEL
LIN {X 0,Y 237.318,Z 1062.504,A -85,B 0,C 180,E1 6466.724,E2 6466.724} C_VEL
LIN {X 0,Y 218.51,Z 1077.264,A -85,B 0,C 180,E1 6463.936,E2 6463.936} C_VEL
LIN {X 0,Y 201.774,Z 1089.067,A -85,B 0,C 180,E1 6460.909,E2 6460.909} C_VEL
LIN {X 0,Y 182.172,Z 1101.537,A -85,B 0,C 180,E1 6456.437,E2 6456.437} C_VEL
LIN {X 0,Y 165.915,Z 1110.836,A -85,B 0,C 180,E1 6451.627,E2 6451.627} C_VEL
LIN {X 0,Y 149.062,Z 1119.735,A -85,B 0,C 180,E1 6444.921,E2 6444.921} C_VEL
LIN {X 0,Y 135.166,Z 1126.469,A -85,B 0,C 180,E1 6437.084,E2 6437.084} C_VEL
LIN {X 0,Y 123.715,Z 1131.976,A -85,B 0,C 180,E1 6427.313,E2 6427.313} C_VEL
LIN {X 0,Y 116.067,Z 1135.665,A -85,B 0,C 180,E1 6416.063,E2 6416.063} C_VEL
LIN {X 0,Y 112.72,Z 1137.667,A -85,B 0,C 180,E1 6405.433,E2 6405.433} C_VEL
LIN {X 0,Y 112.081,Z 1138.454,A -85,B 0,C 180,E1 6395.118,E2 6395.118} C_VEL
LIN {X 0,Y 112.164,Z 1138.251,A -85,B 0,C 180,E1 6388.468,E2 6388.468} C_VEL
LIN {X 0,Y 112.121,Z 1137.418,A -85,B 0,C 180,E1 6380.763,E2 6380.763} C_VEL
LIN {X 0,Y 113.643,Z 1135.288,A -85,B 0,C 180,E1 6370.296,E2 6370.296} C_VEL
LIN {X 0,Y 119.255,Z 1131.008,A -85,B 0,C 180,E1 6358.114,E2 6358.114} C_VEL
LIN {X 0,Y 127.367,Z 1125.966,A -85,B 0,C 180,E1 6348.743,E2 6348.743} C_VEL
LIN {X 0,Y 140.555,Z 1118.213,A -85,B 0,C 180,E1 6339.157,E2 6339.157} C_VEL
LIN {X 0,Y 154.026,Z 1110.079,A -85,B 0,C 180,E1 6332.443,E2 6332.443} C_VEL
LIN {X 0,Y 170.72,Z 1099.491,A -85,B 0,C 180,E1 6326.348,E2 6326.348} C_VEL
LIN {X 0,Y 186.502,Z 1088.518,A -85,B 0,C 180,E1 6321.951,E2 6321.951} C_VEL
LIN {X 0,Y 204.061,Z 1075.339,A -85,B 0,C 180,E1 6318.085,E2 6318.085} C_VEL
LIN {X 0,Y 221.504,Z 1060.63,A -85,B 0,C 180,E1 6314.979,E2 6314.979} C_VEL
LIN {X 0,Y 237.69,Z 1045.66,A -85,B 0,C 180,E1 6312.589,E2 6312.589} C_VEL
LIN {X 0,Y 254.705,Z 1027.951,A -85,B 0,C 180,E1 6310.458,E2 6310.458} C_VEL
LIN {X 0,Y 268.736,Z 1011.704,A -85,B 0,C 180,E1 6308.938,E2 6308.938} C_VEL
LIN {X 0,Y 284.374,Z 991.291,A -85,B 0,C 180,E1 6307.454,E2 6307.454} C_VEL
LIN {X 0,Y 296.342,Z 973.607,A -85,B 0,C 180,E1 6306.444,E2 6306.444} C_VEL
LIN {X 0,Y 309.366,Z 951.808,A -85,B 0,C 180,E1 6305.449,E2 6305.449} C_VEL
LIN {X 0,Y 320.048,Z 930.914,A -85,B 0,C 180,E1 6304.71,E2 6304.71} C_VEL
LIN {X 0,Y 329.811,Z 908.895,A -85,B 0,C 180,E1 6304.103,E2 6304.103} C_VEL
LIN {X 0,Y 338.139,Z 885.891,A -85,B 0,C 180,E1 6303.619,E2 6303.619} C_VEL
LIN {X 0,Y 344.975,Z 862.975,A -85,B 0,C 180,E1 6303.238,E2 6303.238} C_VEL
LIN {X 0,Y 350.504,Z 838.174,A -85,B 0,C 180,E1 6302.893,E2 6302.893} C_VEL
LIN {X 0,Y 354.187,Z 815.025,A -85,B 0,C 180,E1 6302.601,E2 6302.601} C_VEL
LIN {X 0,Y 364.513,Z 727.981,A -85,B 0,C 180,E1 6301.533,E2 6301.533} C_VEL
LIN {X 0,Y 364.292,Z 726.826,A -85,B 0,C 180,E1 6300.315,E2 6300.315} C_VEL
LIN {X 0,Y 364.275,Z 726.821,A -85,B 0,C 180,E1 6296.223,E2 6296.223} C_VEL
LIN {X 0,Y 364.473,Z 728.194,A -85,B 0,C 180,E1 6294.964,E2 6294.964} C_VEL
LIN {X 0,Y 352.96,Z 823.197,A -85,B 0,C 180,E1 6293.833,E2 6293.833} C_VEL
LIN {X 0,Y 348.07,Z 848.885,A -85,B 0,C 180,E1 6293.471,E2 6293.471} C_VEL
LIN {X 0,Y 342.687,Z 869.881,A -85,B 0,C 180,E1 6293.1,E2 6293.1} C_VEL
LIN {X 0,Y 334.302,Z 895.591,A -85,B 0,C 180,E1 6292.509,E2 6292.509} C_VEL
LIN {X 0,Y 326.208,Z 915.847,A -85,B 0,C 180,E1 6291.916,E2 6291.916} C_VEL
LIN {X 0,Y 315.765,Z 938.122,A -85,B 0,C 180,E1 6291.105,E2 6291.105} C_VEL
